LIN {X 0,Y 474.618,Z 134.358,A -85,B 0,C 180,E1 -7419.646,E2 -7419.646} C_VEL
LIN {X 0,Y 474.617,Z 134.363,A -85,B 0,C 180,E1 -7422.934,E2 -7422.934} C_VEL
LIN {X 0,Y 474.606,Z 134.364,A -85,B 0,C 180,E1 -7425.894,E2 -7425.894} C_VEL
LIN {X 0,Y 474.625,Z 134.361,A -85,B 0,C 180,E1 -7429.042,E2 -7429.042} C_VEL
LIN {X 0,Y 474.614,Z 134.364,A -85,B 0,C 180,E1 -7431.704,E2 -7431.704} C_VEL
LIN {X 0,Y 474.628,Z 134.361,A -85,B 0,C 180,E1 -7434.726,E2 -7434.726} C_VEL
LIN {X 0,Y 474.64,Z 134.365,A -85,B 0,C 180,E1 -7437.788,E2 -7437.788} C_VEL
LIN {X 0,Y 474.627,Z 134.362,A -85,B 0,C 180,E1 -7440.885,E2 -7440.885} C_VEL
LIN {X 0,Y 474.666,Z 134.362,A -85,B 0,C 180,E1 -7443.628,E2 -7443.628} C_VEL
LIN {X 0,Y 474.697,Z 134.422,A -85,B 0,C 180,E1 -7444.926,E2 -7444.926} C_VEL
LIN {X 0,Y 475.746,Z 140.895,A -85,B 0,C 180,E1 -7446.335,E2 -7446.335} C_VEL
LIN {X 0,Y 475.555,Z 150.09,A -85,B 0,C 180,E1 -7448.214,E2 -7448.214} C_VEL
LIN {X 0,Y 478.426,Z 164.474,A -85,B 0,C 180,E1 -7448.557,E2 -7448.557} C_VEL
LIN {X 0,Y 478.376,Z 175.483,A -85,B 0,C 180,E1 -7448.726,E2 -7448.726} C_VEL
LIN {X 0,Y 477.685,Z 181.33,A -85,B 0,C 180,E1 -7448.79,E2 -7448.79} C_VEL
LIN {X 0,Y 472.03,Z 200.344,A -85,B 0,C 180,E1 -7448.866,E2 -7448.866} C_VEL
LIN {X 0,Y 471.362,Z 206.19,A -85,B 0,C 180,E1 -7448.932,E2 -7448.932} C_VEL
LIN {X 0,Y 470.901,Z 258.071,A -85,B 0,C 180,E1 -7449.753,E2 -7449.753} C_VEL
LIN {X 0,Y 470.549,Z 271.601,A -85,B 0,C 180,E1 -7450.149,E2 -7450.149} C_VEL
LIN {X 0,Y 470.242,Z 283.825,A -85,B 0,C 180,E1 -7450.685,E2 -7450.685} C_VEL
LIN {X 0,Y 469.795,Z 295.138,A -85,B 0,C 180,E1 -7451.351,E2 -7451.351} C_VEL
LIN {X 0,Y 469.182,Z 306.762,A -85,B 0,C 180,E1 -7452.229,E2 -7452.229} C_VEL
LIN {X 0,Y 468.729,Z 317.2,A -85,B 0,C 180,E1 -7453.224,E2 -7453.224} C_VEL
LIN {X 0,Y 468.335,Z 326.528,A -85,B 0,C 180,E1 -7454.328,E2 -7454.328} C_VEL
LIN {X 0,Y 467.799,Z 335.532,A -85,B 0,C 180,E1 -7455.647,E2 -7455.647} C_VEL
LIN {X 0,Y 467.428,Z 342.757,A -85,B 0,C 180,E1 -7456.965,E2 -7456.965} C_VEL
LIN {X 0,Y 467.168,Z 348.535,A -85,B 0,C 180,E1 -7458.293,E2 -7458.293} C_VEL
LIN {X 0,Y 466.955,Z 352.989,A -85,B 0,C 180,E1 -7459.594,E2 -7459.594} C_VEL
LIN {X 0,Y 466.832,Z 355.353,A -85,B 0,C 180,E1 -7460.467,E2 -7460.467} C_VEL
LIN {X 0,Y 466.795,Z 357.283,A -85,B 0,C 180,E1 -7461.34,E2 -7461.34} C_VEL
LIN {X 0,Y 466.753,Z 358.793,A -85,B 0,C 180,E1 -7462.211,E2 -7462.211} C_VEL
LIN {X 0,Y 466.786,Z 360.292,A -85,B 0,C 180,E1 -7463.571,E2 -7463.571} C_VEL
LIN {X 0,Y 466.71,Z 360.795,A -85,B 0,C 180,E1 -7464.815,E2 -7464.815} C_VEL
LIN {X 0,Y 466.671,Z 360.695,A -85,B 0,C 180,E1 -7465.681,E2 -7465.681} C_VEL
LIN {X 0,Y 466.773,Z 360.159,A -85,B 0,C 180,E1 -7466.546,E2 -7466.546} C_VEL
LIN {X 0,Y 466.71,Z 357.94,A -85,B 0,C 180,E1 -7468.273,E2 -7468.273} C_VEL
LIN {X 0,Y 466.756,Z 355.182,A -85,B 0,C 180,E1 -7469.568,E2 -7469.568} C_VEL
LIN {X 0,Y 466.822,Z 351.423,A -85,B 0,C 180,E1 -7470.862,E2 -7470.862} C_VEL
LIN {X 0,Y 467.123,Z 346.544,A -85,B 0,C 180,E1 -7472.155,E2 -7472.155} C_VEL
LIN {X 0,Y 467.282,Z 340.432,A -85,B 0,C 180,E1 -7473.448,E2 -7473.448} C_VEL
LIN {X 0,Y 467.539,Z 335.515,A -85,B 0,C 180,E1 -7474.31,E2 -7474.31} C_VEL
LIN {X 0,Y 468.082,Z 326.668,A -85,B 0,C 180,E1 -7475.6,E2 -7475.6} C_VEL
LIN {X 0,Y 468.554,Z 317.59,A -85,B 0,C 180,E1 -7476.675,E2 -7476.675} C_VEL
LIN {X 0,Y 469.073,Z 307.492,A -85,B 0,C 180,E1 -7477.64,E2 -7477.64} C_VEL
LIN {X 0,Y 469.554,Z 296.307,A -85,B 0,C 180,E1 -7478.499,E2 -7478.499} C_VEL
LIN {X 0,Y 469.933,Z 284.157,A -85,B 0,C 180,E1 -7479.228,E2 -7479.228} C_VEL
LIN {X 0,Y 470.209,Z 271.377,A -85,B 0,C 180,E1 -7479.788,E2 -7479.788} C_VEL
LIN {X 0,Y 470.485,Z 258.684,A -85,B 0,C 180,E1 -7480.162,E2 -7480.162} C_VEL
LIN {X 0,Y 470.775,Z 232.471,A -85,B 0,C 180,E1 -7480.591,E2 -7480.591} C_VEL
LIN {X 0,Y 471.136,Z 164.035,A -85,B 0,C 180,E1 -7481.638,E2 -7481.638} C_VEL
LIN {X 0,Y 468.426,Z 150.239,A -85,B 0,C 180,E1 -7481.96,E2 -7481.96} C_VEL
LIN {X 0,Y 468.453,Z 139.769,A -85,B 0,C 180,E1 -7484.109,E2 -7484.109} C_VEL
LIN {X 0,Y 467.712,Z 135.226,A -85,B 0,C 180,E1 -7485.133,E2 -7485.133} C_VEL
LIN {X 0,Y 467.614,Z 135.236,A -85,B 0,C 180,E1 -7488.762,E2 -7488.762} C_VEL
LIN {X 0,Y 467.581,Z 135.237,A -85,B 0,C 180,E1 -7491.267,E2 -7491.267} C_VEL
LIN {X 0,Y 467.563,Z 135.244,A -85,B 0,C 180,E1 -7493.943,E2 -7493.943} C_VEL
LIN {X 0,Y 467.612,Z 135.235,A -85,B 0,C 180,E1 -7496.799,E2 -7496.799} C_VEL
LIN {X 0,Y 467.551,Z 135.245,A -85,B 0,C 180,E1 -7499.737,E2 -7499.737} C_VEL
LIN {X 0,Y 467.581,Z 135.238,A -85,B 0,C 180,E1 -7502.757,E2 -7502.757} C_VEL
LIN {X 0,Y 467.55,Z 135.249,A -85,B 0,C 180,E1 -7505.888,E2 -7505.888} C_VEL
LIN {X 0,Y 467.578,Z 135.24,A -85,B 0,C 180,E1 -7509.143,E2 -7509.143} C_VEL
LIN {X 0,Y 467.581,Z 135.239,A -85,B 0,C 180,E1 -7512.566,E2 -7512.566} C_VEL
LIN {X 0,Y 467.56,Z 135.243,A -85,B 0,C 180,E1 -7515.051,E2 -7515.051} C_VEL
LIN {X 0,Y 467.582,Z 135.243,A -85,B 0,C 180,E1 -7517.439,E2 -7517.439} C_VEL
LIN {X 0,Y 467.552,Z 135.244,A -85,B 0,C 180,E1 -7520.852,E2 -7520.852} C_VEL
LIN {X 0,Y 467.55,Z 135.243,A -85,B 0,C 180,E1 -7524.26,E2 -7524.26} C_VEL
LIN {X 0,Y 467.57,Z 135.245,A -85,B 0,C 180,E1 -7527.32,E2 -7527.32} C_VEL
LIN {X 0,Y 467.558,Z 135.244,A -85,B 0,C 180,E1 -7530.667,E2 -7530.667} C_VEL
LIN {X 0,Y 467.576,Z 135.244,A -85,B 0,C 180,E1 -7533.197,E2 -7533.197} C_VEL
LIN {X 0,Y 467.578,Z 135.241,A -85,B 0,C 180,E1 -7536.469,E2 -7536.469} C_VEL
LIN {X 0,Y 467.609,Z 135.237,A -85,B 0,C 180,E1 -7539.776,E2 -7539.776} C_VEL
LIN {X 0,Y 467.575,Z 135.242,A -85,B 0,C 180,E1 -7542.505,E2 -7542.505} C_VEL
LIN {X 0,Y 467.584,Z 135.24,A -85,B 0,C 180,E1 -7545.196,E2 -7545.196} C_VEL
LIN {X 0,Y 467.644,Z 135.234,A -85,B 0,C 180,E1 -7547.854,E2 -7547.854} C_VEL
LIN {X 0,Y 467.653,Z 135.231,A -85,B 0,C 180,E1 -7551.357,E2 -7551.357} C_VEL
LIN {X 0,Y 467.69,Z 135.228,A -85,B 0,C 180,E1 -7553.962,E2 -7553.962} C_VEL
LIN {X 0,Y 467.799,Z 135.214,A -85,B 0,C 180,E1 -7557.417,E2 -7557.417} C_VEL
LIN {X 0,Y 467.836,Z 135.21,A -85,B 0,C 180,E1 -7560,E2 -7560} C_VEL
LIN {X 0,Y 467.8,Z 135.214,A -85,B 0,C 180,E1 -7562.583,E2 -7562.583} C_VEL
LIN {X 0,Y 467.695,Z 135.227,A -85,B 0,C 180,E1 -7566.038,E2 -7566.038} C_VEL
LIN {X 0,Y 467.653,Z 135.231,A -85,B 0,C 180,E1 -7568.643,E2 -7568.643} C_VEL
LIN {X 0,Y 467.644,Z 135.234,A -85,B 0,C 180,E1 -7572.146,E2 -7572.146} C_VEL
LIN {X 0,Y 467.636,Z 135.234,A -85,B 0,C 180,E1 -7575.885,E2 -7575.885} C_VEL
LIN {X 0,Y 467.609,Z 135.238,A -85,B 0,C 180,E1 -7579.308,E2 -7579.308} C_VEL
LIN {X 0,Y 467.519,Z 135.248,A -85,B 0,C 180,E1 -7582.075,E2 -7582.075} C_VEL
LIN {X 0,Y 467.557,Z 135.247,A -85,B 0,C 180,E1 -7584.89,E2 -7584.89} C_VEL
LIN {X 0,Y 467.605,Z 135.237,A -85,B 0,C 180,E1 -7587.77,E2 -7587.77} C_VEL
LIN {X 0,Y 467.557,Z 135.245,A -85,B 0,C 180,E1 -7591.045,E2 -7591.045} C_VEL
LIN {X 0,Y 467.567,Z 135.242,A -85,B 0,C 180,E1 -7594.241,E2 -7594.241} C_VEL
LIN {X 0,Y 467.538,Z 135.245,A -85,B 0,C 180,E1 -7597.187,E2 -7597.187} C_VEL
LIN {X 0,Y 467.566,Z 135.244,A -85,B 0,C 180,E1 -7600.266,E2 -7600.266} C_VEL
LIN {X 0,Y 467.579,Z 135.243,A -85,B 0,C 180,E1 -7602.568,E2 -7602.568} C_VEL
LIN {X 0,Y 467.559,Z 135.242,A -85,B 0,C 180,E1 -7605.054,E2 -7605.054} C_VEL
LIN {X 0,Y 467.583,Z 135.238,A -85,B 0,C 180,E1 -7607.441,E2 -7607.441} C_VEL
LIN {X 0,Y 467.577,Z 135.239,A -85,B 0,C 180,E1 -7610.856,E2 -7610.856} C_VEL
LIN {X 0,Y 467.555,Z 135.246,A -85,B 0,C 180,E1 -7614.262,E2 -7614.262} C_VEL
LIN {X 0,Y 467.578,Z 135.238,A -85,B 0,C 180,E1 -7617.322,E2 -7617.322} C_VEL
LIN {X 0,Y 467.567,Z 135.243,A -85,B 0,C 180,E1 -7620.669,E2 -7620.669} C_VEL
LIN {X 0,Y 467.651,Z 135.252,A -85,B 0,C 180,E1 -7623.714,E2 -7623.714} C_VEL
LIN {X 0,Y 469.785,Z 147.105,A -85,B 0,C 180,E1 -7625.862,E2 -7625.862} C_VEL
LIN {X 0,Y 469.132,Z 164.184,A -85,B 0,C 180,E1 -7628.742,E2 -7628.742} C_VEL
LIN {X 0,Y 468.427,Z 182.92,A -85,B 0,C 180,E1 -7631.862,E2 -7631.862} C_VEL
LIN {X 0,Y 468.193,Z 190.165,A -85,B 0,C 180,E1 -7633.061,E2 -7633.061} C_VEL
LIN {X 0,Y 471.01,Z 210.369,A -85,B 0,C 180,E1 -7633.47,E2 -7633.47} C_VEL
LIN {X 0,Y 470.392,Z 299.136,A -85,B 0,C 180,E1 -7634.844,E2 -7634.844} C_VEL
LIN {X 0,Y 469.994,Z 311.574,A -85,B 0,C 180,E1 -7635.191,E2 -7635.191} C_VEL
LIN {X 0,Y 469.516,Z 325.058,A -85,B 0,C 180,E1 -7635.757,E2 -7635.757} C_VEL
LIN {X 0,Y 469.017,Z 337.151,A -85,B 0,C 180,E1 -7636.46,E2 -7636.46} C_VEL
LIN {X 0,Y 468.525,Z 348.652,A -85,B 0,C 180,E1 -7637.324,E2 -7637.324} C_VEL
LIN {X 0,Y 468.07,Z 359.11,A -85,B 0,C 180,E1 -7638.306,E2 -7638.306} C_VEL
LIN {X 0,Y 467.602,Z 368.448,A -85,B 0,C 180,E1 -7639.391,E2 -7639.391} C_VEL
LIN {X 0,Y 467.207,Z 377.51,A -85,B 0,C 180,E1 -7640.695,E2 -7640.695} C_VEL
LIN {X 0,Y 466.979,Z 384.813,A -85,B 0,C 180,E1 -7641.999,E2 -7641.999} C_VEL
LIN {X 0,Y 466.827,Z 389.743,A -85,B 0,C 180,E1 -7643.083,E2 -7643.083} C_VEL
LIN {X 0,Y 466.749,Z 394.534,A -85,B 0,C 180,E1 -7644.384,E2 -7644.384} C_VEL
LIN {X 0,Y 466.647,Z 398.195,A -85,B 0,C 180,E1 -7645.682,E2 -7645.682} C_VEL
LIN {X 0,Y 466.73,Z 400.093,A -85,B 0,C 180,E1 -7646.548,E2 -7646.548} C_VEL
LIN {X 0,Y 466.685,Z 401.519,A -85,B 0,C 180,E1 -7647.411,E2 -7647.411} C_VEL
LIN {X 0,Y 466.662,Z 402.532,A -85,B 0,C 180,E1 -7648.275,E2 -7648.275} C_VEL
LIN {X 0,Y 466.611,Z 403.387,A -85,B 0,C 180,E1 -7650.001,E2 -7650.001} C_VEL
LIN {X 0,Y 466.627,Z 403.192,A -85,B 0,C 180,E1 -7650.864,E2 -7650.864} C_VEL
LIN {X 0,Y 466.662,Z 402.596,A -85,B 0,C 180,E1 -7651.727,E2 -7651.727} C_VEL
LIN {X 0,Y 466.685,Z 401.61,A -85,B 0,C 180,E1 -7652.59,E2 -7652.59} C_VEL
LIN {X 0,Y 466.7,Z 400.226,A -85,B 0,C 180,E1 -7653.454,E2 -7653.454} C_VEL
LIN {X 0,Y 466.687,Z 397.304,A -85,B 0,C 180,E1 -7654.752,E2 -7654.752} C_VEL
LIN {X 0,Y 466.719,Z 393.351,A -85,B 0,C 180,E1 -7656.051,E2 -7656.051} C_VEL
LIN {X 0,Y 466.883,Z 388.271,A -85,B 0,C 180,E1 -7657.352,E2 -7657.352} C_VEL
LIN {X 0,Y 467.112,Z 381.892,A -85,B 0,C 180,E1 -7658.654,E2 -7658.654} C_VEL
LIN {X 0,Y 467.425,Z 373.921,A -85,B 0,C 180,E1 -7659.958,E2 -7659.958} C_VEL
LIN {X 0,Y 467.878,Z 365.819,A -85,B 0,C 180,E1 -7661.042,E2 -7661.042} C_VEL
LIN {X 0,Y 468.324,Z 355.951,A -85,B 0,C 180,E1 -7662.128,E2 -7662.128} C_VEL
LIN {X 0,Y 468.809,Z 344.917,A -85,B 0,C 180,E1 -7663.106,E2 -7663.106} C_VEL
LIN {X 0,Y 469.352,Z 334.121,A -85,B 0,C 180,E1 -7663.862,E2 -7663.862} C_VEL
LIN {X 0,Y 469.895,Z 321.117,A -85,B 0,C 180,E1 -7664.564,E2 -7664.564} C_VEL
LIN {X 0,Y 470.368,Z 308.577,A -85,B 0,C 180,E1 -7665.047,E2 -7665.047} C_VEL
LIN {X 0,Y 470.732,Z 295.474,A -85,B 0,C 180,E1 -7665.368,E2 -7665.368} C_VEL
LIN {X 0,Y 471.218,Z 209.135,A -85,B 0,C 180,E1 -7666.708,E2 -7666.708} C_VEL
LIN {X 0,Y 468.32,Z 189.921,A -85,B 0,C 180,E1 -7667.145,E2 -7667.145} C_VEL
LIN {X 0,Y 468.918,Z 173.306,A -85,B 0,C 180,E1 -7669.937,E2 -7669.937} C_VEL
LIN {X 0,Y 469.766,Z 155.911,A -85,B 0,C 180,E1 -7672.891,E2 -7672.891} C_VEL
LIN {X 0,Y 469.986,Z 147.08,A -85,B 0,C 180,E1 -7674.421,E2 -7674.421} C_VEL
LIN {X 0,Y 467.614,Z 135.239,A -85,B 0,C 180,E1 -7676.68,E2 -7676.68} C_VEL
LIN {X 0,Y 467.55,Z 135.251,A -85,B 0,C 180,E1 -7679.739,E2 -7679.739} C_VEL
LIN {X 0,Y 467.586,Z 135.24,A -85,B 0,C 180,E1 -7682.759,E2 -7682.759} C_VEL
LIN {X 0,Y 467.553,Z 135.246,A -85,B 0,C 180,E1 -7685.89,E2 -7685.89} C_VEL
LIN {X 0,Y 467.557,Z 135.242,A -85,B 0,C 180,E1 -7689.148,E2 -7689.148} C_VEL
LIN {X 0,Y 467.575,Z 135.243,A -85,B 0,C 180,E1 -7691.403,E2 -7691.403} C_VEL
LIN {X 0,Y 467.567,Z 135.242,A -85,B 0,C 180,E1 -7695.052,E2 -7695.052} C_VEL
LIN {X 0,Y 467.568,Z 135.24,A -85,B 0,C 180,E1 -7698.596,E2 -7698.596} C_VEL
LIN {X 0,Y 467.564,Z 135.241,A -85,B 0,C 180,E1 -7701.955,E2 -7701.955} C_VEL
LIN {X 0,Y 467.559,Z 135.247,A -85,B 0,C 180,E1 -7705.167,E2 -7705.167} C_VEL
LIN {X 0,Y 467.58,Z 135.239,A -85,B 0,C 180,E1 -7708.26,E2 -7708.26} C_VEL
LIN {X 0,Y 467.544,Z 135.245,A -85,B 0,C 180,E1 -7711.248,E2 -7711.248} C_VEL
LIN {X 0,Y 467.578,Z 135.24,A -85,B 0,C 180,E1 -7714.401,E2 -7714.401} C_VEL
LIN {X 0,Y 467.568,Z 135.243,A -85,B 0,C 180,E1 -7716.995,E2 -7716.995} C_VEL
LIN {X 0,Y 467.61,Z 135.231,A -85,B 0,C 180,E1 -7719.777,E2 -7719.777} C_VEL
LIN {X 0,Y 467.564,Z 135.245,A -85,B 0,C 180,E1 -7722.505,E2 -7722.505} C_VEL
LIN {X 0,Y 467.586,Z 135.232,A -85,B 0,C 180,E1 -7725.196,E2 -7725.196} C_VEL
LIN {X 0,Y 467.64,Z 135.231,A -85,B 0,C 180,E1 -7727.854,E2 -7727.854} C_VEL
LIN {X 0,Y 467.628,Z 135.226,A -85,B 0,C 180,E1 -7731.356,E2 -7731.356} C_VEL
LIN {X 0,Y 467.698,Z 135.228,A -85,B 0,C 180,E1 -7733.962,E2 -7733.962} C_VEL
LIN {X 0,Y 467.808,Z 135.205,A -85,B 0,C 180,E1 -7737.417,E2 -7737.417} C_VEL
LIN {X 0,Y 467.848,Z 135.21,A -85,B 0,C 180,E1 -7740,E2 -7740} C_VEL
LIN {X 0,Y 467.811,Z 135.203,A -85,B 0,C 180,E1 -7742.583,E2 -7742.583} C_VEL
LIN {X 0,Y 467.7,Z 135.226,A -85,B 0,C 180,E1 -7746.038,E2 -7746.038} C_VEL
LIN {X 0,Y 467.663,Z 135.221,A -85,B 0,C 180,E1 -7748.643,E2 -7748.643} C_VEL
LIN {X 0,Y 467.656,Z 135.228,A -85,B 0,C 180,E1 -7752.146,E2 -7752.146} C_VEL
LIN {X 0,Y 467.649,Z 135.23,A -85,B 0,C 180,E1 -7755.885,E2 -7755.885} C_VEL
LIN {X 0,Y 467.621,Z 135.234,A -85,B 0,C 180,E1 -7759.308,E2 -7759.308} C_VEL
LIN {X 0,Y 467.531,Z 135.244,A -85,B 0,C 180,E1 -7762.074,E2 -7762.074} C_VEL
LIN {X 0,Y 467.569,Z 135.24,A -85,B 0,C 180,E1 -7764.89,E2 -7764.89} C_VEL
LIN {X 0,Y 467.581,Z 135.236,A -85,B 0,C 180,E1 -7767.772,E2 -7767.772} C_VEL
LIN {X 0,Y 467.568,Z 135.243,A -85,B 0,C 180,E1 -7771.045,E2 -7771.045} C_VEL
LIN {X 0,Y 467.579,Z 135.239,A -85,B 0,C 180,E1 -7774.24,E2 -7774.24} C_VEL
LIN {X 0,Y 467.549,Z 135.243,A -85,B 0,C 180,E1 -7777.186,E2 -7777.186} C_VEL
LIN {X 0,Y 467.577,Z 135.238,A -85,B 0,C 180,E1 -7780.265,E2 -7780.265} C_VEL
LIN {X 0,Y 467.59,Z 135.239,A -85,B 0,C 180,E1 -7782.567,E2 -7782.567} C_VEL
LIN {X 0,Y 467.568,Z 135.239,A -85,B 0,C 180,E1 -7785.053,E2 -7785.053} C_VEL
LIN {X 0,Y 467.576,Z 135.242,A -85,B 0,C 180,E1 -7788.597,E2 -7788.597} C_VEL
LIN {X 0,Y 467.564,Z 135.24,A -85,B 0,C 180,E1 -7791.409,E2 -7791.409} C_VEL
LIN {X 0,Y 467.564,Z 135.245,A -85,B 0,C 180,E1 -7794.261,E2 -7794.261} C_VEL
LIN {X 0,Y 467.586,Z 135.239,A -85,B 0,C 180,E1 -7797.321,E2 -7797.321} C_VEL
LIN {X 0,Y 467.573,Z 135.241,A -85,B 0,C 180,E1 -7800.668,E2 -7800.668} C_VEL
LIN {X 0,Y 467.621,Z 135.238,A -85,B 0,C 180,E1 -7803.2,E2 -7803.2} C_VEL
LIN {X 0,Y 467.657,Z 135.37,A -85,B 0,C 180,E1 -7804.742,E2 -7804.742} C_VEL
LIN {X 0,Y 468.808,Z 142.348,A -85,B 0,C 180,E1 -7806.277,E2 -7806.277} C_VEL
LIN {X 0,Y 468.64,Z 150.392,A -85,B 0,C 180,E1 -7807.937,E2 -7807.937} C_VEL
LIN {X 0,Y 471.683,Z 165.079,A -85,B 0,C 180,E1 -7808.299,E2 -7808.299} C_VEL
LIN {X 0,Y 471.362,Z 206.19,A -85,B 0,C 180,E1 -7808.932,E2 -7808.932} C_VEL
LIN {X 0,Y 470.683,Z 212.035,A -85,B 0,C 180,E1 -7808.997,E2 -7808.997} C_VEL
LIN {X 0,Y 464.988,Z 231.034,A -85,B 0,C 180,E1 -7809.074,E2 -7809.074} C_VEL
LIN {X 0,Y 464.348,Z 236.877,A -85,B 0,C 180,E1 -7809.142,E2 -7809.142} C_VEL
LIN {X 0,Y 464.074,Z 259.518,A -85,B 0,C 180,E1 -7809.528,E2 -7809.528} C_VEL
LIN {X 0,Y 463.761,Z 272.58,A -85,B 0,C 180,E1 -7809.929,E2 -7809.929} C_VEL
LIN {X 0,Y 463.436,Z 283.39,A -85,B 0,C 180,E1 -7810.41,E2 -7810.41} C_VEL
LIN {X 0,Y 462.994,Z 294.64,A -85,B 0,C 180,E1 -7811.067,E2 -7811.067} C_VEL
LIN {X 0,Y 462.342,Z 306.423,A -85,B 0,C 180,E1 -7811.957,E2 -7811.957} C_VEL
LIN {X 0,Y 461.893,Z 316.974,A -85,B 0,C 180,E1 -7812.968,E2 -7812.968} C_VEL
LIN {X 0,Y 461.402,Z 326.432,A -85,B 0,C 180,E1 -7814.087,E2 -7814.087} C_VEL
LIN {X 0,Y 460.835,Z 335.506,A -85,B 0,C 180,E1 -7815.425,E2 -7815.425} C_VEL
LIN {X 0,Y 460.428,Z 342.792,A -85,B 0,C 180,E1 -7816.763,E2 -7816.763} C_VEL
LIN {X 0,Y 460.136,Z 348.828,A -85,B 0,C 180,E1 -7818.161,E2 -7818.161} C_VEL
LIN {X 0,Y 459.924,Z 353.147,A -85,B 0,C 180,E1 -7819.433,E2 -7819.433} C_VEL
LIN {X 0,Y 459.764,Z 355.539,A -85,B 0,C 180,E1 -7820.319,E2 -7820.319} C_VEL
LIN {X 0,Y 459.732,Z 357.49,A -85,B 0,C 180,E1 -7821.206,E2 -7821.206} C_VEL
LIN {X 0,Y 459.669,Z 359.028,A -85,B 0,C 180,E1 -7822.09,E2 -7822.09} C_VEL
LIN {X 0,Y 459.715,Z 360.645,A -85,B 0,C 180,E1 -7823.569,E2 -7823.569} C_VEL
LIN {X 0,Y 459.643,Z 361.108,A -85,B 0,C 180,E1 -7824.736,E2 -7824.736} C_VEL
LIN {X 0,Y 459.582,Z 361.034,A -85,B 0,C 180,E1 -7825.614,E2 -7825.614} C_VEL
LIN {X 0,Y 459.699,Z 360.535,A -85,B 0,C 180,E1 -7826.493,E2 -7826.493} C_VEL
LIN {X 0,Y 459.647,Z 358.356,A -85,B 0,C 180,E1 -7828.247,E2 -7828.247} C_VEL
LIN {X 0,Y 459.669,Z 355.644,A -85,B 0,C 180,E1 -7829.561,E2 -7829.561} C_VEL
LIN {X 0,Y 459.745,Z 351.931,A -85,B 0,C 180,E1 -7830.875,E2 -7830.875} C_VEL
LIN {X 0,Y 460.067,Z 347.1,A -85,B 0,C 180,E1 -7832.188,E2 -7832.188} C_VEL
LIN {X 0,Y 460.234,Z 341.041,A -85,B 0,C 180,E1 -7833.501,E2 -7833.501} C_VEL
LIN {X 0,Y 460.707,Z 333.493,A -85,B 0,C 180,E1 -7834.812,E2 -7834.812} C_VEL
LIN {X 0,Y 461.228,Z 324.015,A -85,B 0,C 180,E1 -7836.122,E2 -7836.122} C_VEL
LIN {X 0,Y 461.803,Z 314.239,A -85,B 0,C 180,E1 -7837.212,E2 -7837.212} C_VEL
LIN {X 0,Y 462.333,Z 303.269,A -85,B 0,C 180,E1 -7838.192,E2 -7838.192} C_VEL
LIN {X 0,Y 462.81,Z 291.752,A -85,B 0,C 180,E1 -7839.003,E2 -7839.003} C_VEL
LIN {X 0,Y 463.181,Z 279.605,A -85,B 0,C 180,E1 -7839.662,E2 -7839.662} C_VEL
LIN {X 0,Y 463.481,Z 266.996,A -85,B 0,C 180,E1 -7840.152,E2 -7840.152} C_VEL
LIN {X 0,Y 463.673,Z 253.728,A -85,B 0,C 180,E1 -7840.479,E2 -7840.479} C_VEL
LIN {X 0,Y 464.349,Z 165.216,A -85,B 0,C 180,E1 -7841.853,E2 -7841.853} C_VEL
LIN {X 0,Y 461.447,Z 150.541,A -85,B 0,C 180,E1 -7842.199,E2 -7842.199} C_VEL
LIN {X 0,Y 461.511,Z 141.339,A -85,B 0,C 180,E1 -7844.101,E2 -7844.101} C_VEL
LIN {X 0,Y 460.668,Z 136.104,A -85,B 0,C 180,E1 -7845.257,E2 -7845.257} C_VEL
LIN {X 0,Y 460.568,Z 136.112,A -85,B 0,C 180,E1 -7848.899,E2 -7848.899} C_VEL
LIN {X 0,Y 460.516,Z 136.118,A -85,B 0,C 180,E1 -7851.484,E2 -7851.484} C_VEL
LIN {X 0,Y 460.531,Z 136.121,A -85,B 0,C 180,E1 -7854.332,E2 -7854.332} C_VEL
LIN {X 0,Y 460.57,Z 136.112,A -85,B 0,C 180,E1 -7857.243,E2 -7857.243} C_VEL
LIN {X 0,Y 460.508,Z 136.123,A -85,B 0,C 180,E1 -7860.239,E2 -7860.239} C_VEL
LIN {X 0,Y 460.526,Z 136.118,A -85,B 0,C 180,E1 -7863.324,E2 -7863.324} C_VEL
LIN {X 0,Y 460.472,Z 136.125,A -85,B 0,C 180,E1 -7866.528,E2 -7866.528} C_VEL
LIN {X 0,Y 460.553,Z 136.119,A -85,B 0,C 180,E1 -7869.858,E2 -7869.858} C_VEL
LIN {X 0,Y 460.507,Z 136.121,A -85,B 0,C 180,E1 -7872.899,E2 -7872.899} C_VEL
LIN {X 0,Y 460.501,Z 136.124,A -85,B 0,C 180,E1 -7875.83,E2 -7875.83} C_VEL
LIN {X 0,Y 460.523,Z 136.119,A -85,B 0,C 180,E1 -7878.988,E2 -7878.988} C_VEL
LIN {X 0,Y 460.511,Z 136.123,A -85,B 0,C 180,E1 -7881.265,E2 -7881.265} C_VEL
LIN {X 0,Y 460.5,Z 136.123,A -85,B 0,C 180,E1 -7884.553,E2 -7884.553} C_VEL
LIN {X 0,Y 460.52,Z 136.12,A -85,B 0,C 180,E1 -7887.714,E2 -7887.714} C_VEL
LIN {X 0,Y 460.528,Z 136.119,A -85,B 0,C 180,E1 -7890.768,E2 -7890.768} C_VEL
LIN {X 0,Y 460.531,Z 136.118,A -85,B 0,C 180,E1 -7893.733,E2 -7893.733} C_VEL
LIN {X 0,Y 460.531,Z 136.119,A -85,B 0,C 180,E1 -7896.623,E2 -7896.623} C_VEL
LIN {X 0,Y 460.538,Z 136.118,A -85,B 0,C 180,E1 -7899.452,E2 -7899.452} C_VEL
LIN {X 0,Y 460.528,Z 136.12,A -85,B 0,C 180,E1 -7902.229,E2 -7902.229} C_VEL
LIN {X 0,Y 460.545,Z 136.119,A -85,B 0,C 180,E1 -7904.964,E2 -7904.964} C_VEL
LIN {X 0,Y 460.596,Z 136.112,A -85,B 0,C 180,E1 -7908.559,E2 -7908.559} C_VEL
LIN {X 0,Y 460.604,Z 136.11,A -85,B 0,C 180,E1 -7911.223,E2 -7911.223} C_VEL
LIN {X 0,Y 460.656,Z 136.104,A -85,B 0,C 180,E1 -7913.869,E2 -7913.869} C_VEL
LIN {X 0,Y 460.743,Z 136.093,A -85,B 0,C 180,E1 -7917.377,E2 -7917.377} C_VEL
LIN {X 0,Y 460.805,Z 136.085,A -85,B 0,C 180,E1 -7920,E2 -7920} C_VEL
LIN {X 0,Y 460.744,Z 136.093,A -85,B 0,C 180,E1 -7922.623,E2 -7922.623} C_VEL
LIN {X 0,Y 460.661,Z 136.103,A -85,B 0,C 180,E1 -7926.13,E2 -7926.13} C_VEL
LIN {X 0,Y 460.604,Z 136.109,A -85,B 0,C 180,E1 -7928.777,E2 -7928.777} C_VEL
LIN {X 0,Y 460.584,Z 136.112,A -85,B 0,C 180,E1 -7932.435,E2 -7932.435} C_VEL
LIN {X 0,Y 460.589,Z 136.112,A -85,B 0,C 180,E1 -7935.998,E2 -7935.998} C_VEL
LIN {X 0,Y 460.555,Z 136.116,A -85,B 0,C 180,E1 -7939.616,E2 -7939.616} C_VEL
LIN {X 0,Y 460.495,Z 136.123,A -85,B 0,C 180,E1 -7942.429,E2 -7942.429} C_VEL
LIN {X 0,Y 460.535,Z 136.118,A -85,B 0,C 180,E1 -7945.797,E2 -7945.797} C_VEL
LIN {X 0,Y 460.539,Z 136.117,A -85,B 0,C 180,E1 -7948.234,E2 -7948.234} C_VEL
LIN {X 0,Y 460.51,Z 136.121,A -85,B 0,C 180,E1 -7951.283,E2 -7951.283} C_VEL
LIN {X 0,Y 460.513,Z 136.123,A -85,B 0,C 180,E1 -7954.505,E2 -7954.505} C_VEL
LIN {X 0,Y 460.492,Z 136.122,A -85,B 0,C 180,E1 -7957.624,E2 -7957.624} C_VEL
LIN {X 0,Y 460.531,Z 136.12,A -85,B 0,C 180,E1 -7960.27,E2 -7960.27} C_VEL
LIN {X 0,Y 460.489,Z 136.122,A -85,B 0,C 180,E1 -7963.377,E2 -7963.377} C_VEL
LIN {X 0,Y 460.492,Z 136.124,A -85,B 0,C 180,E1 -7966.626,E2 -7966.626} C_VEL
LIN {X 0,Y 460.536,Z 136.117,A -85,B 0,C 180,E1 -7969.732,E2 -7969.732} C_VEL
LIN {X 0,Y 460.494,Z 136.123,A -85,B 0,C 180,E1 -7972.525,E2 -7972.525} C_VEL
LIN {X 0,Y 460.542,Z 136.116,A -85,B 0,C 180,E1 -7975.625,E2 -7975.625} C_VEL
LIN {X 0,Y 460.534,Z 136.118,A -85,B 0,C 180,E1 -7978.746,E2 -7978.746} C_VEL
LIN {X 0,Y 460.579,Z 136.115,A -85,B 0,C 180,E1 -7982.255,E2 -7982.255} C_VEL
LIN {X 0,Y 460.618,Z 136.308,A -85,B 0,C 180,E1 -7983.556,E2 -7983.556} C_VEL
LIN {X 0,Y 462.777,Z 147.763,A -85,B 0,C 180,E1 -7985.671,E2 -7985.671} C_VEL
LIN {X 0,Y 462.29,Z 161.486,A -85,B 0,C 180,E1 -7988.027,E2 -7988.027} C_VEL
LIN {X 0,Y 461.531,Z 181.108,A -85,B 0,C 180,E1 -7991.352,E2 -7991.352} C_VEL
LIN {X 0,Y 461.196,Z 189.853,A -85,B 0,C 180,E1 -7992.821,E2 -7992.821} C_VEL
LIN {X 0,Y 464.146,Z 211.204,A -85,B 0,C 180,E1 -7993.258,E2 -7993.258} C_VEL
LIN {X 0,Y 463.508,Z 299.121,A -85,B 0,C 180,E1 -7994.642,E2 -7994.642} C_VEL
LIN {X 0,Y 463.061,Z 312.224,A -85,B 0,C 180,E1 -7995.021,E2 -7995.021} C_VEL
LIN {X 0,Y 462.627,Z 324.325,A -85,B 0,C 180,E1 -7995.541,E2 -7995.541} C_VEL
LIN {X 0,Y 462.057,Z 336.54,A -85,B 0,C 180,E1 -7996.253,E2 -7996.253} C_VEL
LIN {X 0,Y 461.533,Z 348.094,A -85,B 0,C 180,E1 -7997.129,E2 -7997.129} C_VEL
LIN {X 0,Y 461.052,Z 358.597,A -85,B 0,C 180,E1 -7998.126,E2 -7998.126} C_VEL
LIN {X 0,Y 460.594,Z 367.984,A -85,B 0,C 180,E1 -7999.228,E2 -7999.228} C_VEL
LIN {X 0,Y 460.163,Z 377.07,A -85,B 0,C 180,E1 -8000.551,E2 -8000.551} C_VEL
LIN {X 0,Y 459.907,Z 384.394,A -85,B 0,C 180,E1 -8001.875,E2 -8001.875} C_VEL
LIN {X 0,Y 459.739,Z 389.343,A -85,B 0,C 180,E1 -8002.976,E2 -8002.976} C_VEL
LIN {X 0,Y 459.645,Z 394.152,A -85,B 0,C 180,E1 -8004.297,E2 -8004.297} C_VEL
LIN {X 0,Y 459.564,Z 397.829,A -85,B 0,C 180,E1 -8005.616,E2 -8005.616} C_VEL
LIN {X 0,Y 459.625,Z 399.735,A -85,B 0,C 180,E1 -8006.494,E2 -8006.494} C_VEL
LIN {X 0,Y 459.607,Z 401.174,A -85,B 0,C 180,E1 -8007.372,E2 -8007.372} C_VEL
LIN {X 0,Y 459.559,Z 402.822,A -85,B 0,C 180,E1 -8009.125,E2 -8009.125} C_VEL
LIN {X 0,Y 459.542,Z 403.062,A -85,B 0,C 180,E1 -8010.001,E2 -8010.001} C_VEL
LIN {X 0,Y 459.56,Z 402.879,A -85,B 0,C 180,E1 -8010.877,E2 -8010.877} C_VEL
LIN {X 0,Y 459.605,Z 401.308,A -85,B 0,C 180,E1 -8012.63,E2 -8012.63} C_VEL
LIN {X 0,Y 459.595,Z 399.93,A -85,B 0,C 180,E1 -8013.508,E2 -8013.508} C_VEL
LIN {X 0,Y 459.614,Z 397.022,A -85,B 0,C 180,E1 -8014.825,E2 -8014.825} C_VEL
LIN {X 0,Y 459.635,Z 392.408,A -85,B 0,C 180,E1 -8016.343,E2 -8016.343} C_VEL
LIN {X 0,Y 459.869,Z 386.034,A -85,B 0,C 180,E1 -8017.906,E2 -8017.906} C_VEL
LIN {X 0,Y 460.15,Z 379.195,A -85,B 0,C 180,E1 -8019.229,E2 -8019.229} C_VEL
LIN {X 0,Y 460.531,Z 370.693,A -85,B 0,C 180,E1 -8020.553,E2 -8020.553} C_VEL
LIN {X 0,Y 461.042,Z 361.963,A -85,B 0,C 180,E1 -8021.653,E2 -8021.653} C_VEL
LIN {X 0,Y 461.532,Z 351.797,A -85,B 0,C 180,E1 -8022.703,E2 -8022.703} C_VEL
LIN {X 0,Y 462.142,Z 340.565,A -85,B 0,C 180,E1 -8023.634,E2 -8023.634} C_VEL
LIN {X 0,Y 462.749,Z 328.631,A -85,B 0,C 180,E1 -8024.401,E2 -8024.401} C_VEL
LIN {X 0,Y 463.292,Z 316.226,A -85,B 0,C 180,E1 -8025.001,E2 -8025.001} C_VEL
LIN {X 0,Y 463.743,Z 303.43,A -85,B 0,C 180,E1 -8025.436,E2 -8025.436} C_VEL
LIN {X 0,Y 463.992,Z 289.871,A -85,B 0,C 180,E1 -8025.709,E2 -8025.709} C_VEL
LIN {X 0,Y 464.516,Z 210.176,A -85,B 0,C 180,E1 -8026.956,E2 -8026.956} C_VEL
LIN {X 0,Y 461.362,Z 189.617,A -85,B 0,C 180,E1 -8027.429,E2 -8027.429} C_VEL
LIN {X 0,Y 462.007,Z 173.117,A -85,B 0,C 180,E1 -8030.248,E2 -8030.248} C_VEL
LIN {X 0,Y 462.859,Z 157.071,A -85,B 0,C 180,E1 -8033.016,E2 -8033.016} C_VEL
LIN {X 0,Y 463.137,Z 149.036,A -85,B 0,C 180,E1 -8034.427,E2 -8034.427} C_VEL
LIN {X 0,Y 460.727,Z 136.92,A -85,B 0,C 180,E1 -8036.744,E2 -8036.744} C_VEL
LIN {X 0,Y 460.584,Z 136.114,A -85,B 0,C 180,E1 -8036.937,E2 -8036.937} C_VEL
LIN {X 0,Y 460.51,Z 136.128,A -85,B 0,C 180,E1 -8040.241,E2 -8040.241} C_VEL
LIN {X 0,Y 460.532,Z 136.12,A -85,B 0,C 180,E1 -8043.325,E2 -8043.325} C_VEL
LIN {X 0,Y 460.475,Z 136.122,A -85,B 0,C 180,E1 -8046.53,E2 -8046.53} C_VEL
LIN {X 0,Y 460.522,Z 136.121,A -85,B 0,C 180,E1 -8049.864,E2 -8049.864} C_VEL
LIN {X 0,Y 460.494,Z 136.12,A -85,B 0,C 180,E1 -8052.898,E2 -8052.898} C_VEL
LIN {X 0,Y 460.506,Z 136.122,A -85,B 0,C 180,E1 -8055.831,E2 -8055.831} C_VEL
LIN {X 0,Y 460.521,Z 136.121,A -85,B 0,C 180,E1 -8058.987,E2 -8058.987} C_VEL
LIN {X 0,Y 460.501,Z 136.12,A -85,B 0,C 180,E1 -8062.377,E2 -8062.377} C_VEL
LIN {X 0,Y 460.537,Z 136.117,A -85,B 0,C 180,E1 -8065.623,E2 -8065.623} C_VEL
LIN {X 0,Y 460.538,Z 136.12,A -85,B 0,C 180,E1 -8068.745,E2 -8068.745} C_VEL
LIN {X 0,Y 460.531,Z 136.116,A -85,B 0,C 180,E1 -8072.266,E2 -8072.266} C_VEL
LIN {X 0,Y 460.522,Z 136.122,A -85,B 0,C 180,E1 -8074.703,E2 -8074.703} C_VEL
LIN {X 0,Y 460.503,Z 136.119,A -85,B 0,C 180,E1 -8077.571,E2 -8077.571} C_VEL
LIN {X 0,Y 460.561,Z 136.112,A -85,B 0,C 180,E1 -8080.384,E2 -8080.384} C_VEL
LIN {X 0,Y 460.567,Z 136.114,A -85,B 0,C 180,E1 -8084.058,E2 -8084.058} C_VEL
LIN {X 0,Y 460.601,Z 136.106,A -85,B 0,C 180,E1 -8087.666,E2 -8087.666} C_VEL
LIN {X 0,Y 460.583,Z 136.103,A -85,B 0,C 180,E1 -8091.223,E2 -8091.223} C_VEL
LIN {X 0,Y 460.664,Z 136.103,A -85,B 0,C 180,E1 -8093.87,E2 -8093.87} C_VEL
LIN {X 0,Y 460.752,Z 136.083,A -85,B 0,C 180,E1 -8097.377,E2 -8097.377} C_VEL
LIN {X 0,Y 460.817,Z 136.086,A -85,B 0,C 180,E1 -8100,E2 -8100} C_VEL
LIN {X 0,Y 460.755,Z 136.082,A -85,B 0,C 180,E1 -8102.623,E2 -8102.623} C_VEL
LIN {X 0,Y 460.666,Z 136.101,A -85,B 0,C 180,E1 -8106.131,E2 -8106.131} C_VEL
LIN {X 0,Y 460.614,Z 136.099,A -85,B 0,C 180,E1 -8108.777,E2 -8108.777} C_VEL
LIN {X 0,Y 460.597,Z 136.107,A -85,B 0,C 180,E1 -8112.435,E2 -8112.435} C_VEL
LIN {X 0,Y 460.602,Z 136.108,A -85,B 0,C 180,E1 -8115.998,E2 -8115.998} C_VEL
LIN {X 0,Y 460.568,Z 136.111,A -85,B 0,C 180,E1 -8119.616,E2 -8119.616} C_VEL
LIN {X 0,Y 460.508,Z 136.119,A -85,B 0,C 180,E1 -8122.429,E2 -8122.429} C_VEL
LIN {X 0,Y 460.548,Z 136.114,A -85,B 0,C 180,E1 -8125.797,E2 -8125.797} C_VEL
LIN {X 0,Y 460.528,Z 136.115,A -85,B 0,C 180,E1 -8128.235,E2 -8128.235} C_VEL
LIN {X 0,Y 460.521,Z 136.119,A -85,B 0,C 180,E1 -8131.283,E2 -8131.283} C_VEL
LIN {X 0,Y 460.525,Z 136.121,A -85,B 0,C 180,E1 -8134.504,E2 -8134.504} C_VEL
LIN {X 0,Y 460.503,Z 136.119,A -85,B 0,C 180,E1 -8137.623,E2 -8137.623} C_VEL
LIN {X 0,Y 460.541,Z 136.114,A -85,B 0,C 180,E1 -8140.269,E2 -8140.269} C_VEL
LIN {X 0,Y 460.501,Z 136.119,A -85,B 0,C 180,E1 -8143.376,E2 -8143.376} C_VEL
LIN {X 0,Y 460.511,Z 136.122,A -85,B 0,C 180,E1 -8146.626,E2 -8146.626} C_VEL
LIN {X 0,Y 460.54,Z 136.118,A -85,B 0,C 180,E1 -8149.731,E2 -8149.731} C_VEL
LIN {X 0,Y 460.503,Z 136.122,A -85,B 0,C 180,E1 -8152.524,E2 -8152.524} C_VEL
LIN {X 0,Y 460.55,Z 136.118,A -85,B 0,C 180,E1 -8155.624,E2 -8155.624} C_VEL
LIN {X 0,Y 460.542,Z 136.116,A -85,B 0,C 180,E1 -8158.744,E2 -8158.744} C_VEL
LIN {X 0,Y 460.585,Z 136.115,A -85,B 0,C 180,E1 -8162.254,E2 -8162.254} C_VEL
LIN {X 0,Y 460.601,Z 136.137,A -85,B 0,C 180,E1 -8164.506,E2 -8164.506} C_VEL
LIN {X 0,Y 461.76,Z 142.609,A -85,B 0,C 180,E1 -8165.952,E2 -8165.952} C_VEL
LIN {X 0,Y 461.748,Z 150.618,A -85,B 0,C 180,E1 -8167.634,E2 -8167.634} C_VEL
LIN {X 0,Y 464.91,Z 165.279,A -85,B 0,C 180,E1 -8168.023,E2 -8168.023} C_VEL
LIN {X 0,Y 464.348,Z 236.877,A -85,B 0,C 180,E1 -8169.142,E2 -8169.142} C_VEL
LIN {X 0,Y 463.667,Z 240.808,A -85,B 0,C 180,E1 -8169.177,E2 -8169.177} C_VEL
LIN {X 0,Y 457.964,Z 253.099,A -85,B 0,C 180,E1 -8169.152,E2 -8169.152} C_VEL
LIN {X 0,Y 457.389,Z 257.002,A -85,B 0,C 180,E1 -8169.204,E2 -8169.204} C_VEL
LIN {X 0,Y 457.035,Z 270.027,A -85,B 0,C 180,E1 -8169.569,E2 -8169.569} C_VEL
LIN {X 0,Y 456.635,Z 282.983,A -85,B 0,C 180,E1 -8170.127,E2 -8170.127} C_VEL
LIN {X 0,Y 456.223,Z 294.095,A -85,B 0,C 180,E1 -8170.775,E2 -8170.775} C_VEL
LIN {X 0,Y 455.634,Z 304.792,A -85,B 0,C 180,E1 -8171.566,E2 -8171.566} C_VEL
LIN {X 0,Y 455.05,Z 315.682,A -85,B 0,C 180,E1 -8172.588,E2 -8172.588} C_VEL
LIN {X 0,Y 454.588,Z 324.406,A -85,B 0,C 180,E1 -8173.593,E2 -8173.593} C_VEL
LIN {X 0,Y 454.078,Z 332.658,A -85,B 0,C 180,E1 -8174.744,E2 -8174.744} C_VEL
LIN {X 0,Y 453.579,Z 340.59,A -85,B 0,C 180,E1 -8176.103,E2 -8176.103} C_VEL
LIN {X 0,Y 453.212,Z 346.889,A -85,B 0,C 180,E1 -8177.461,E2 -8177.461} C_VEL
LIN {X 0,Y 452.944,Z 351.879,A -85,B 0,C 180,E1 -8178.816,E2 -8178.816} C_VEL
LIN {X 0,Y 452.707,Z 355.728,A -85,B 0,C 180,E1 -8180.167,E2 -8180.167} C_VEL
LIN {X 0,Y 452.662,Z 357.701,A -85,B 0,C 180,E1 -8181.067,E2 -8181.067} C_VEL
LIN {X 0,Y 452.604,Z 359.26,A -85,B 0,C 180,E1 -8181.966,E2 -8181.966} C_VEL
LIN {X 0,Y 452.632,Z 361.002,A -85,B 0,C 180,E1 -8183.581,E2 -8183.581} C_VEL
LIN {X 0,Y 452.578,Z 361.42,A -85,B 0,C 180,E1 -8184.653,E2 -8184.653} C_VEL
LIN {X 0,Y 452.499,Z 361.367,A -85,B 0,C 180,E1 -8185.545,E2 -8185.545} C_VEL
LIN {X 0,Y 452.608,Z 360.909,A -85,B 0,C 180,E1 -8186.438,E2 -8186.438} C_VEL
LIN {X 0,Y 452.555,Z 358.772,A -85,B 0,C 180,E1 -8188.219,E2 -8188.219} C_VEL
LIN {X 0,Y 452.586,Z 356.102,A -85,B 0,C 180,E1 -8189.554,E2 -8189.554} C_VEL
LIN {X 0,Y 452.67,Z 352.433,A -85,B 0,C 180,E1 -8190.889,E2 -8190.889} C_VEL
LIN {X 0,Y 453.011,Z 347.65,A -85,B 0,C 180,E1 -8192.222,E2 -8192.222} C_VEL
LIN {X 0,Y 453.187,Z 341.643,A -85,B 0,C 180,E1 -8193.556,E2 -8193.556} C_VEL
LIN {X 0,Y 453.681,Z 334.163,A -85,B 0,C 180,E1 -8194.887,E2 -8194.887} C_VEL
LIN {X 0,Y 454.16,Z 326.521,A -85,B 0,C 180,E1 -8195.995,E2 -8195.995} C_VEL
LIN {X 0,Y 454.68,Z 317.21,A -85,B 0,C 180,E1 -8197.102,E2 -8197.102} C_VEL
LIN {X 0,Y 455.249,Z 306.877,A -85,B 0,C 180,E1 -8198.097,E2 -8198.097} C_VEL
LIN {X 0,Y 455.798,Z 295.483,A -85,B 0,C 180,E1 -8198.975,E2 -8198.975} C_VEL
LIN {X 0,Y 456.16,Z 284.026,A -85,B 0,C 180,E1 -8199.663,E2 -8199.663} C_VEL
LIN {X 0,Y 456.472,Z 271.286,A -85,B 0,C 180,E1 -8200.225,E2 -8200.225} C_VEL
LIN {X 0,Y 456.787,Z 258.22,A -85,B 0,C 180,E1 -8200.61,E2 -8200.61} C_VEL
LIN {X 0,Y 457.504,Z 166.082,A -85,B 0,C 180,E1 -8202.08,E2 -8202.08} C_VEL
LIN {X 0,Y 454.496,Z 150.838,A -85,B 0,C 180,E1 -8202.445,E2 -8202.445} C_VEL
LIN {X 0,Y 454.574,Z 142.941,A -85,B 0,C 180,E1 -8204.092,E2 -8204.092} C_VEL
LIN {X 0,Y 453.599,Z 136.984,A -85,B 0,C 180,E1 -8205.429,E2 -8205.429} C_VEL
LIN {X 0,Y 453.518,Z 136.99,A -85,B 0,C 180,E1 -8209.038,E2 -8209.038} C_VEL
LIN {X 0,Y 453.477,Z 136.997,A -85,B 0,C 180,E1 -8211.835,E2 -8211.835} C_VEL
LIN {X 0,Y 453.5,Z 136.993,A -85,B 0,C 180,E1 -8214.734,E2 -8214.734} C_VEL
LIN {X 0,Y 453.53,Z 136.993,A -85,B 0,C 180,E1 -8217.958,E2 -8217.958} C_VEL
LIN {X 0,Y 453.463,Z 136.998,A -85,B 0,C 180,E1 -8221.524,E2 -8221.524} C_VEL
LIN {X 0,Y 453.484,Z 136.995,A -85,B 0,C 180,E1 -8224.776,E2 -8224.776} C_VEL
LIN {X 0,Y 453.46,Z 136.999,A -85,B 0,C 180,E1 -8228.31,E2 -8228.31} C_VEL
LIN {X 0,Y 453.489,Z 136.995,A -85,B 0,C 180,E1 -8230.608,E2 -8230.608} C_VEL
LIN {X 0,Y 453.449,Z 137.001,A -85,B 0,C 180,E1 -8233.243,E2 -8233.243} C_VEL
LIN {X 0,Y 453.455,Z 137.002,A -85,B 0,C 180,E1 -8235.777,E2 -8235.777} C_VEL
LIN {X 0,Y 453.472,Z 136.997,A -85,B 0,C 180,E1 -8238.208,E2 -8238.208} C_VEL
LIN {X 0,Y 453.479,Z 136.996,A -85,B 0,C 180,E1 -8240.793,E2 -8240.793} C_VEL
LIN {X 0,Y 453.445,Z 137.001,A -85,B 0,C 180,E1 -8243.916,E2 -8243.916} C_VEL
LIN {X 0,Y 453.47,Z 137,A -85,B 0,C 180,E1 -8247.15,E2 -8247.15} C_VEL
LIN {X 0,Y 453.464,Z 136.999,A -85,B 0,C 180,E1 -8250.267,E2 -8250.267} C_VEL
LIN {X 0,Y 453.522,Z 136.992,A -85,B 0,C 180,E1 -8252.296,E2 -8252.296} C_VEL
LIN {X 0,Y 453.481,Z 136.999,A -85,B 0,C 180,E1 -8255.263,E2 -8255.263} C_VEL
LIN {X 0,Y 453.469,Z 136.998,A -85,B 0,C 180,E1 -8258.414,E2 -8258.414} C_VEL
LIN {X 0,Y 453.511,Z 136.996,A -85,B 0,C 180,E1 -8261.008,E2 -8261.008} C_VEL
LIN {X 0,Y 453.526,Z 136.993,A -85,B 0,C 180,E1 -8263.893,E2 -8263.893} C_VEL
LIN {X 0,Y 453.552,Z 136.988,A -85,B 0,C 180,E1 -8267.471,E2 -8267.471} C_VEL
LIN {X 0,Y 453.57,Z 136.986,A -85,B 0,C 180,E1 -8271.086,E2 -8271.086} C_VEL
LIN {X 0,Y 453.624,Z 136.981,A -85,B 0,C 180,E1 -8273.774,E2 -8273.774} C_VEL
LIN {X 0,Y 453.69,Z 136.972,A -85,B 0,C 180,E1 -8277.336,E2 -8277.336} C_VEL
LIN {X 0,Y 453.754,Z 136.963,A -85,B 0,C 180,E1 -8280,E2 -8280} C_VEL
LIN {X 0,Y 453.691,Z 136.971,A -85,B 0,C 180,E1 -8282.664,E2 -8282.664} C_VEL
LIN {X 0,Y 453.628,Z 136.979,A -85,B 0,C 180,E1 -8286.226,E2 -8286.226} C_VEL
LIN {X 0,Y 453.57,Z 136.986,A -85,B 0,C 180,E1 -8288.914,E2 -8288.914} C_VEL
LIN {X 0,Y 453.552,Z 136.988,A -85,B 0,C 180,E1 -8292.529,E2 -8292.529} C_VEL
LIN {X 0,Y 453.532,Z 136.991,A -85,B 0,C 180,E1 -8296.196,E2 -8296.196} C_VEL
LIN {X 0,Y 453.505,Z 136.997,A -85,B 0,C 180,E1 -8299.04,E2 -8299.04} C_VEL
LIN {X 0,Y 453.464,Z 136.999,A -85,B 0,C 180,E1 -8301.837,E2 -8301.837} C_VEL
LIN {X 0,Y 453.48,Z 136.999,A -85,B 0,C 180,E1 -8304.736,E2 -8304.736} C_VEL
LIN {X 0,Y 453.518,Z 136.992,A -85,B 0,C 180,E1 -8307.959,E2 -8307.959} C_VEL
LIN {X 0,Y 453.455,Z 136.999,A -85,B 0,C 180,E1 -8311.526,E2 -8311.526} C_VEL
LIN {X 0,Y 453.473,Z 137,A -85,B 0,C 180,E1 -8314.777,E2 -8314.777} C_VEL
LIN {X 0,Y 453.452,Z 137.002,A -85,B 0,C 180,E1 -8318.313,E2 -8318.313} C_VEL
LIN {X 0,Y 453.486,Z 136.999,A -85,B 0,C 180,E1 -8320.61,E2 -8320.61} C_VEL
LIN {X 0,Y 453.445,Z 137,A -85,B 0,C 180,E1 -8323.245,E2 -8323.245} C_VEL
LIN {X 0,Y 453.457,Z 136.999,A -85,B 0,C 180,E1 -8325.78,E2 -8325.78} C_VEL
LIN {X 0,Y 453.473,Z 137.001,A -85,B 0,C 180,E1 -8328.21,E2 -8328.21} C_VEL
LIN {X 0,Y 453.51,Z 136.992,A -85,B 0,C 180,E1 -8330.791,E2 -8330.791} C_VEL
LIN {X 0,Y 453.449,Z 137.002,A -85,B 0,C 180,E1 -8333.918,E2 -8333.918} C_VEL
LIN {X 0,Y 453.479,Z 136.994,A -85,B 0,C 180,E1 -8337.152,E2 -8337.152} C_VEL
LIN {X 0,Y 453.472,Z 137.002,A -85,B 0,C 180,E1 -8340.27,E2 -8340.27} C_VEL
LIN {X 0,Y 453.57,Z 137.093,A -85,B 0,C 180,E1 -8343.345,E2 -8343.345} C_VEL
LIN {X 0,Y 455.847,Z 149.205,A -85,B 0,C 180,E1 -8345.617,E2 -8345.617} C_VEL
LIN {X 0,Y 455.181,Z 165.714,A -85,B 0,C 180,E1 -8348.489,E2 -8348.489} C_VEL
LIN {X 0,Y 454.38,Z 184.698,A -85,B 0,C 180,E1 -8351.748,E2 -8351.748} C_VEL
LIN {X 0,Y 454.217,Z 189.481,A -85,B 0,C 180,E1 -8352.565,E2 -8352.565} C_VEL
LIN {X 0,Y 457.296,Z 212.314,A -85,B 0,C 180,E1 -8353.046,E2 -8353.046} C_VEL
LIN {X 0,Y 456.644,Z 297.896,A -85,B 0,C 180,E1 -8354.405,E2 -8354.405} C_VEL
LIN {X 0,Y 456.177,Z 310.536,A -85,B 0,C 180,E1 -8354.761,E2 -8354.761} C_VEL
LIN {X 0,Y 455.721,Z 323.563,A -85,B 0,C 180,E1 -8355.317,E2 -8355.317} C_VEL
LIN {X 0,Y 455.128,Z 335.911,A -85,B 0,C 180,E1 -8356.039,E2 -8356.039} C_VEL
LIN {X 0,Y 454.576,Z 347.317,A -85,B 0,C 180,E1 -8356.911,E2 -8356.911} C_VEL
LIN {X 0,Y 453.995,Z 358.065,A -85,B 0,C 180,E1 -8357.938,E2 -8357.938} C_VEL
LIN {X 0,Y 453.594,Z 367.509,A -85,B 0,C 180,E1 -8359.06,E2 -8359.06} C_VEL
LIN {X 0,Y 453.127,Z 376.622,A -85,B 0,C 180,E1 -8360.403,E2 -8360.403} C_VEL
LIN {X 0,Y 452.831,Z 383.968,A -85,B 0,C 180,E1 -8361.747,E2 -8361.747} C_VEL
LIN {X 0,Y 452.667,Z 388.938,A -85,B 0,C 180,E1 -8362.866,E2 -8362.866} C_VEL
LIN {X 0,Y 452.543,Z 393.763,A -85,B 0,C 180,E1 -8364.207,E2 -8364.207} C_VEL
LIN {X 0,Y 452.486,Z 397.46,A -85,B 0,C 180,E1 -8365.547,E2 -8365.547} C_VEL
LIN {X 0,Y 452.521,Z 399.372,A -85,B 0,C 180,E1 -8366.439,E2 -8366.439} C_VEL
LIN {X 0,Y 452.53,Z 400.826,A -85,B 0,C 180,E1 -8367.33,E2 -8367.33} C_VEL
LIN {X 0,Y 452.494,Z 402.489,A -85,B 0,C 180,E1 -8369.111,E2 -8369.111} C_VEL
LIN {X 0,Y 452.475,Z 402.737,A -85,B 0,C 180,E1 -8370.001,E2 -8370.001} C_VEL
LIN {X 0,Y 452.494,Z 402.567,A -85,B 0,C 180,E1 -8370.891,E2 -8370.891} C_VEL
LIN {X 0,Y 452.527,Z 401.008,A -85,B 0,C 180,E1 -8372.671,E2 -8372.671} C_VEL
LIN {X 0,Y 452.492,Z 399.637,A -85,B 0,C 180,E1 -8373.563,E2 -8373.563} C_VEL
LIN {X 0,Y 452.541,Z 396.744,A -85,B 0,C 180,E1 -8374.901,E2 -8374.901} C_VEL
LIN {X 0,Y 452.554,Z 392.53,A -85,B 0,C 180,E1 -8376.332,E2 -8376.332} C_VEL
LIN {X 0,Y 452.733,Z 387.775,A -85,B 0,C 180,E1 -8377.583,E2 -8377.583} C_VEL
LIN {X 0,Y 452.984,Z 381.447,A -85,B 0,C 180,E1 -8378.926,E2 -8378.926} C_VEL
LIN {X 0,Y 453.362,Z 373.535,A -85,B 0,C 180,E1 -8380.27,E2 -8380.27} C_VEL
LIN {X 0,Y 454.002,Z 363.705,A -85,B 0,C 180,E1 -8381.61,E2 -8381.61} C_VEL
LIN {X 0,Y 454.449,Z 354.499,A -85,B 0,C 180,E1 -8382.631,E2 -8382.631} C_VEL
LIN {X 0,Y 455.07,Z 343.374,A -85,B 0,C 180,E1 -8383.623,E2 -8383.623} C_VEL
LIN {X 0,Y 455.654,Z 332.373,A -85,B 0,C 180,E1 -8384.402,E2 -8384.402} C_VEL
LIN {X 0,Y 456.24,Z 320.2,A -85,B 0,C 180,E1 -8385.067,E2 -8385.067} C_VEL
LIN {X 0,Y 456.74,Z 307.508,A -85,B 0,C 180,E1 -8385.565,E2 -8385.565} C_VEL
LIN {X 0,Y 457.177,Z 294.143,A -85,B 0,C 180,E1 -8385.893,E2 -8385.893} C_VEL
LIN {X 0,Y 457.737,Z 210.718,A -85,B 0,C 180,E1 -8387.224,E2 -8387.224} C_VEL
LIN {X 0,Y 454.414,Z 189.273,A -85,B 0,C 180,E1 -8387.731,E2 -8387.731} C_VEL
LIN {X 0,Y 455.1,Z 172.935,A -85,B 0,C 180,E1 -8390.569,E2 -8390.569} C_VEL
LIN {X 0,Y 456.063,Z 155.561,A -85,B 0,C 180,E1 -8393.62,E2 -8393.62} C_VEL
LIN {X 0,Y 456.138,Z 149.975,A -85,B 0,C 180,E1 -8394.625,E2 -8394.625} C_VEL
LIN {X 0,Y 453.76,Z 138.098,A -85,B 0,C 180,E1 -8396.939,E2 -8396.939} C_VEL
LIN {X 0,Y 453.514,Z 136.995,A -85,B 0,C 180,E1 -8397.204,E2 -8397.204} C_VEL
LIN {X 0,Y 453.471,Z 137.005,A -85,B 0,C 180,E1 -8399.784,E2 -8399.784} C_VEL
LIN {X 0,Y 453.493,Z 136.997,A -85,B 0,C 180,E1 -8403.189,E2 -8403.189} C_VEL
LIN {X 0,Y 453.453,Z 136.998,A -85,B 0,C 180,E1 -8406.299,E2 -8406.299} C_VEL
LIN {X 0,Y 453.466,Z 136.998,A -85,B 0,C 180,E1 -8409.453,E2 -8409.453} C_VEL
LIN {X 0,Y 453.461,Z 136.999,A -85,B 0,C 180,E1 -8411.932,E2 -8411.932} C_VEL
LIN {X 0,Y 453.484,Z 137,A -85,B 0,C 180,E1 -8415.472,E2 -8415.472} C_VEL
LIN {X 0,Y 453.461,Z 136.997,A -85,B 0,C 180,E1 -8418.207,E2 -8418.207} C_VEL
LIN {X 0,Y 453.449,Z 137.001,A -85,B 0,C 180,E1 -8420.801,E2 -8420.801} C_VEL
LIN {X 0,Y 453.454,Z 136.999,A -85,B 0,C 180,E1 -8423.917,E2 -8423.917} C_VEL
LIN {X 0,Y 453.478,Z 137,A -85,B 0,C 180,E1 -8427.151,E2 -8427.151} C_VEL
LIN {X 0,Y 453.461,Z 136.997,A -85,B 0,C 180,E1 -8430.267,E2 -8430.267} C_VEL
LIN {X 0,Y 453.455,Z 136.999,A -85,B 0,C 180,E1 -8433.291,E2 -8433.291} C_VEL
LIN {X 0,Y 453.492,Z 136.995,A -85,B 0,C 180,E1 -8436.238,E2 -8436.238} C_VEL
LIN {X 0,Y 453.474,Z 136.994,A -85,B 0,C 180,E1 -8439.117,E2 -8439.117} C_VEL
LIN {X 0,Y 453.484,Z 136.992,A -85,B 0,C 180,E1 -8441.943,E2 -8441.943} C_VEL
LIN {X 0,Y 453.516,Z 136.988,A -85,B 0,C 180,E1 -8444.726,E2 -8444.726} C_VEL
LIN {X 0,Y 453.564,Z 136.982,A -85,B 0,C 180,E1 -8447.471,E2 -8447.471} C_VEL
LIN {X 0,Y 453.553,Z 136.979,A -85,B 0,C 180,E1 -8451.086,E2 -8451.086} C_VEL
LIN {X 0,Y 453.633,Z 136.977,A -85,B 0,C 180,E1 -8453.774,E2 -8453.774} C_VEL
LIN {X 0,Y 453.699,Z 136.962,A -85,B 0,C 180,E1 -8457.337,E2 -8457.337} C_VEL
LIN {X 0,Y 453.766,Z 136.964,A -85,B 0,C 180,E1 -8460,E2 -8460} C_VEL
LIN {X 0,Y 453.702,Z 136.96,A -85,B 0,C 180,E1 -8462.664,E2 -8462.664} C_VEL
LIN {X 0,Y 453.634,Z 136.976,A -85,B 0,C 180,E1 -8466.226,E2 -8466.226} C_VEL
LIN {X 0,Y 453.581,Z 136.976,A -85,B 0,C 180,E1 -8468.914,E2 -8468.914} C_VEL
LIN {X 0,Y 453.565,Z 136.983,A -85,B 0,C 180,E1 -8472.529,E2 -8472.529} C_VEL
LIN {X 0,Y 453.545,Z 136.986,A -85,B 0,C 180,E1 -8476.196,E2 -8476.196} C_VEL
LIN {X 0,Y 453.518,Z 136.992,A -85,B 0,C 180,E1 -8479.039,E2 -8479.039} C_VEL
LIN {X 0,Y 453.476,Z 136.995,A -85,B 0,C 180,E1 -8481.836,E2 -8481.836} C_VEL
LIN {X 0,Y 453.494,Z 136.992,A -85,B 0,C 180,E1 -8484.736,E2 -8484.736} C_VEL
LIN {X 0,Y 453.508,Z 136.989,A -85,B 0,C 180,E1 -8487.953,E2 -8487.953} C_VEL
LIN {X 0,Y 453.477,Z 137,A -85,B 0,C 180,E1 -8490.76,E2 -8490.76} C_VEL
LIN {X 0,Y 453.47,Z 136.995,A -85,B 0,C 180,E1 -8493.914,E2 -8493.914} C_VEL
LIN {X 0,Y 453.454,Z 136.998,A -85,B 0,C 180,E1 -8497.19,E2 -8497.19} C_VEL
LIN {X 0,Y 453.496,Z 136.986,A -85,B 0,C 180,E1 -8500.609,E2 -8500.609} C_VEL
LIN {X 0,Y 453.457,Z 136.997,A -85,B 0,C 180,E1 -8503.244,E2 -8503.244} C_VEL
LIN {X 0,Y 453.463,Z 136.997,A -85,B 0,C 180,E1 -8505.778,E2 -8505.778} C_VEL
LIN {X 0,Y 453.497,Z 136.993,A -85,B 0,C 180,E1 -8509.409,E2 -8509.409} C_VEL
LIN {X 0,Y 453.456,Z 136.998,A -85,B 0,C 180,E1 -8512.81,E2 -8512.81} C_VEL
LIN {X 0,Y 453.481,Z 137,A -85,B 0,C 180,E1 -8516.087,E2 -8516.087} C_VEL
LIN {X 0,Y 453.481,Z 136.996,A -85,B 0,C 180,E1 -8519.24,E2 -8519.24} C_VEL
LIN {X 0,Y 453.54,Z 136.993,A -85,B 0,C 180,E1 -8522.297,E2 -8522.297} C_VEL
LIN {X 0,Y 453.555,Z 137.029,A -85,B 0,C 180,E1 -8524.286,E2 -8524.286} C_VEL
LIN {X 0,Y 454.899,Z 144.796,A -85,B 0,C 180,E1 -8526.038,E2 -8526.038} C_VEL
LIN {X 0,Y 454.829,Z 151.028,A -85,B 0,C 180,E1 -8527.355,E2 -8527.355} C_VEL
LIN {X 0,Y 458.208,Z 166.924,A -85,B 0,C 180,E1 -8527.764,E2 -8527.764} C_VEL
LIN {X 0,Y 457.389,Z 257.002,A -85,B 0,C 180,E1 -8529.204,E2 -8529.204} C_VEL
LIN {X 0,Y 456.884,Z 262.791,A -85,B 0,C 180,E1 -8529.322,E2 -8529.322} C_VEL
LIN {X 0,Y 454.006,Z 272.132,A -85,B 0,C 180,E1 -8529.515,E2 -8529.515} C_VEL
LIN {X 0,Y 450.773,Z 281.254,A -85,B 0,C 180,E1 -8529.797,E2 -8529.797} C_VEL
LIN {X 0,Y 449.725,Z 286.709,A -85,B 0,C 180,E1 -8530.056,E2 -8530.056} C_VEL
LIN {X 0,Y 449.166,Z 298.514,A -85,B 0,C 180,E1 -8530.817,E2 -8530.817} C_VEL
LIN {X 0,Y 448.488,Z 309.679,A -85,B 0,C 180,E1 -8531.735,E2 -8531.735} C_VEL
LIN {X 0,Y 447.868,Z 320.486,A -85,B 0,C 180,E1 -8532.867,E2 -8532.867} C_VEL
LIN {X 0,Y 447.392,Z 329.537,A -85,B 0,C 180,E1 -8534.043,E2 -8534.043} C_VEL
LIN {X 0,Y 446.844,Z 336.835,A -85,B 0,C 180,E1 -8535.191,E2 -8535.191} C_VEL
LIN {X 0,Y 446.367,Z 343.989,A -85,B 0,C 180,E1 -8536.571,E2 -8536.571} C_VEL
LIN {X 0,Y 446.117,Z 349.065,A -85,B 0,C 180,E1 -8537.789,E2 -8537.789} C_VEL
LIN {X 0,Y 445.823,Z 353.447,A -85,B 0,C 180,E1 -8539.095,E2 -8539.095} C_VEL
LIN {X 0,Y 445.652,Z 355.92,A -85,B 0,C 180,E1 -8540.01,E2 -8540.01} C_VEL
LIN {X 0,Y 445.581,Z 357.915,A -85,B 0,C 180,E1 -8540.924,E2 -8540.924} C_VEL
LIN {X 0,Y 445.527,Z 359.494,A -85,B 0,C 180,E1 -8541.837,E2 -8541.837} C_VEL
LIN {X 0,Y 445.552,Z 360.662,A -85,B 0,C 180,E1 -8542.75,E2 -8542.75} C_VEL
LIN {X 0,Y 445.532,Z 361.391,A -85,B 0,C 180,E1 -8543.66,E2 -8543.66} C_VEL
LIN {X 0,Y 445.493,Z 361.734,A -85,B 0,C 180,E1 -8544.568,E2 -8544.568} C_VEL
LIN {X 0,Y 445.504,Z 361.276,A -85,B 0,C 180,E1 -8546.381,E2 -8546.381} C_VEL
LIN {X 0,Y 445.502,Z 360.426,A -85,B 0,C 180,E1 -8547.287,E2 -8547.287} C_VEL
LIN {X 0,Y 445.477,Z 357.549,A -85,B 0,C 180,E1 -8549.095,E2 -8549.095} C_VEL
LIN {X 0,Y 445.644,Z 354.255,A -85,B 0,C 180,E1 -8550.451,E2 -8550.451} C_VEL
LIN {X 0,Y 445.734,Z 349.916,A -85,B 0,C 180,E1 -8551.806,E2 -8551.806} C_VEL
LIN {X 0,Y 446.091,Z 344.387,A -85,B 0,C 180,E1 -8553.16,E2 -8553.16} C_VEL
LIN {X 0,Y 446.45,Z 337.497,A -85,B 0,C 180,E1 -8554.514,E2 -8554.514} C_VEL
LIN {X 0,Y 447.063,Z 328.853,A -85,B 0,C 180,E1 -8555.864,E2 -8555.864} C_VEL
LIN {X 0,Y 447.564,Z 320.021,A -85,B 0,C 180,E1 -8556.989,E2 -8556.989} C_VEL
LIN {X 0,Y 448.167,Z 310.307,A -85,B 0,C 180,E1 -8557.999,E2 -8557.999} C_VEL
LIN {X 0,Y 448.664,Z 299.629,A -85,B 0,C 180,E1 -8558.898,E2 -8558.898} C_VEL
LIN {X 0,Y 449.119,Z 288.283,A -85,B 0,C 180,E1 -8559.648,E2 -8559.648} C_VEL
LIN {X 0,Y 449.533,Z 275.175,A -85,B 0,C 180,E1 -8560.3,E2 -8560.3} C_VEL
LIN {X 0,Y 449.841,Z 263,A -85,B 0,C 180,E1 -8560.719,E2 -8560.719} C_VEL
LIN {X 0,Y 449.98,Z 247.603,A -85,B 0,C 180,E1 -8561.029,E2 -8561.029} C_VEL
LIN {X 0,Y 450.723,Z 167.187,A -85,B 0,C 180,E1 -8562.307,E2 -8562.307} C_VEL
LIN {X 0,Y 447.515,Z 151.128,A -85,B 0,C 180,E1 -8562.7,E2 -8562.7} C_VEL
LIN {X 0,Y 447.528,Z 143.481,A -85,B 0,C 180,E1 -8564.319,E2 -8564.319} C_VEL
LIN {X 0,Y 446.545,Z 137.864,A -85,B 0,C 180,E1 -8565.608,E2 -8565.608} C_VEL
LIN {X 0,Y 446.469,Z 137.867,A -85,B 0,C 180,E1 -8569.302,E2 -8569.302} C_VEL
LIN {X 0,Y 446.419,Z 137.88,A -85,B 0,C 180,E1 -8572.198,E2 -8572.198} C_VEL
LIN {X 0,Y 446.443,Z 137.871,A -85,B 0,C 180,E1 -8575.152,E2 -8575.152} C_VEL
LIN {X 0,Y 446.483,Z 137.872,A -85,B 0,C 180,E1 -8578.177,E2 -8578.177} C_VEL
LIN {X 0,Y 446.417,Z 137.878,A -85,B 0,C 180,E1 -8581.774,E2 -8581.774} C_VEL
LIN {X 0,Y 446.426,Z 137.875,A -85,B 0,C 180,E1 -8584.522,E2 -8584.522} C_VEL
LIN {X 0,Y 446.412,Z 137.879,A -85,B 0,C 180,E1 -8588.078,E2 -8588.078} C_VEL
LIN {X 0,Y 446.422,Z 137.875,A -85,B 0,C 180,E1 -8590.916,E2 -8590.916} C_VEL
LIN {X 0,Y 446.394,Z 137.882,A -85,B 0,C 180,E1 -8593.845,E2 -8593.845} C_VEL
LIN {X 0,Y 446.39,Z 137.879,A -85,B 0,C 180,E1 -8596.403,E2 -8596.403} C_VEL
LIN {X 0,Y 446.42,Z 137.876,A -85,B 0,C 180,E1 -8599.081,E2 -8599.081} C_VEL
LIN {X 0,Y 446.399,Z 137.879,A -85,B 0,C 180,E1 -8602.12,E2 -8602.12} C_VEL
LIN {X 0,Y 446.414,Z 137.88,A -85,B 0,C 180,E1 -8605.475,E2 -8605.475} C_VEL
LIN {X 0,Y 446.406,Z 137.878,A -85,B 0,C 180,E1 -8608.699,E2 -8608.699} C_VEL
LIN {X 0,Y 446.475,Z 137.87,A -85,B 0,C 180,E1 -8611.82,E2 -8611.82} C_VEL
LIN {X 0,Y 446.426,Z 137.876,A -85,B 0,C 180,E1 -8614.846,E2 -8614.846} C_VEL
LIN {X 0,Y 446.437,Z 137.875,A -85,B 0,C 180,E1 -8618.245,E2 -8618.245} C_VEL
LIN {X 0,Y 446.435,Z 137.875,A -85,B 0,C 180,E1 -8621.648,E2 -8621.648} C_VEL
LIN {X 0,Y 446.465,Z 137.871,A -85,B 0,C 180,E1 -8624.478,E2 -8624.478} C_VEL
LIN {X 0,Y 446.504,Z 137.866,A -85,B 0,C 180,E1 -8628.193,E2 -8628.193} C_VEL
LIN {X 0,Y 446.518,Z 137.866,A -85,B 0,C 180,E1 -8630.944,E2 -8630.944} C_VEL
LIN {X 0,Y 446.594,Z 137.857,A -85,B 0,C 180,E1 -8633.675,E2 -8633.675} C_VEL
LIN {X 0,Y 446.639,Z 137.85,A -85,B 0,C 180,E1 -8637.294,E2 -8637.294} C_VEL
LIN {X 0,Y 446.705,Z 137.841,A -85,B 0,C 180,E1 -8640,E2 -8640} C_VEL
LIN {X 0,Y 446.64,Z 137.85,A -85,B 0,C 180,E1 -8642.706,E2 -8642.706} C_VEL
LIN {X 0,Y 446.597,Z 137.856,A -85,B 0,C 180,E1 -8646.324,E2 -8646.324} C_VEL
LIN {X 0,Y 446.518,Z 137.866,A -85,B 0,C 180,E1 -8649.056,E2 -8649.056} C_VEL
LIN {X 0,Y 446.509,Z 137.866,A -85,B 0,C 180,E1 -8652.73,E2 -8652.73} C_VEL
LIN {X 0,Y 446.476,Z 137.869,A -85,B 0,C 180,E1 -8656.46,E2 -8656.46} C_VEL
LIN {X 0,Y 446.456,Z 137.873,A -85,B 0,C 180,E1 -8659.304,E2 -8659.304} C_VEL
LIN {X 0,Y 446.405,Z 137.878,A -85,B 0,C 180,E1 -8662.2,E2 -8662.2} C_VEL
LIN {X 0,Y 446.425,Z 137.877,A -85,B 0,C 180,E1 -8665.154,E2 -8665.154} C_VEL
LIN {X 0,Y 446.475,Z 137.869,A -85,B 0,C 180,E1 -8668.179,E2 -8668.179} C_VEL
LIN {X 0,Y 446.408,Z 137.877,A -85,B 0,C 180,E1 -8671.775,E2 -8671.775} C_VEL
LIN {X 0,Y 446.414,Z 137.88,A -85,B 0,C 180,E1 -8674.524,E2 -8674.524} C_VEL
LIN {X 0,Y 446.404,Z 137.878,A -85,B 0,C 180,E1 -8678.08,E2 -8678.08} C_VEL
LIN {X 0,Y 446.419,Z 137.876,A -85,B 0,C 180,E1 -8680.919,E2 -8680.919} C_VEL
LIN {X 0,Y 446.391,Z 137.879,A -85,B 0,C 180,E1 -8683.847,E2 -8683.847} C_VEL
LIN {X 0,Y 446.391,Z 137.883,A -85,B 0,C 180,E1 -8686.405,E2 -8686.405} C_VEL
LIN {X 0,Y 446.421,Z 137.874,A -85,B 0,C 180,E1 -8689.084,E2 -8689.084} C_VEL
LIN {X 0,Y 446.41,Z 137.879,A -85,B 0,C 180,E1 -8691.922,E2 -8691.922} C_VEL
LIN {X 0,Y 446.424,Z 137.874,A -85,B 0,C 180,E1 -8695.478,E2 -8695.478} C_VEL
LIN {X 0,Y 446.412,Z 137.878,A -85,B 0,C 180,E1 -8698.701,E2 -8698.701} C_VEL
LIN {X 0,Y 446.482,Z 137.873,A -85,B 0,C 180,E1 -8701.823,E2 -8701.823} C_VEL
LIN {X 0,Y 446.52,Z 137.894,A -85,B 0,C 180,E1 -8703.13,E2 -8703.13} C_VEL
LIN {X 0,Y 448.706,Z 149.192,A -85,B 0,C 180,E1 -8705.291,E2 -8705.291} C_VEL
LIN {X 0,Y 448.884,Z 152.979,A -85,B 0,C 180,E1 -8705.98,E2 -8705.98} C_VEL
LIN {X 0,Y 447.967,Z 170.669,A -85,B 0,C 180,E1 -8709.09,E2 -8709.09} C_VEL
LIN {X 0,Y 447.223,Z 188.549,A -85,B 0,C 180,E1 -8712.204,E2 -8712.204} C_VEL
LIN {X 0,Y 447.205,Z 189.157,A -85,B 0,C 180,E1 -8712.309,E2 -8712.309} C_VEL
LIN {X 0,Y 450.454,Z 213.931,A -85,B 0,C 180,E1 -8712.836,E2 -8712.836} C_VEL
LIN {X 0,Y 449.775,Z 297.793,A -85,B 0,C 180,E1 -8714.19,E2 -8714.19} C_VEL
LIN {X 0,Y 449.26,Z 311.121,A -85,B 0,C 180,E1 -8714.578,E2 -8714.578} C_VEL
LIN {X 0,Y 448.764,Z 323.913,A -85,B 0,C 180,E1 -8715.142,E2 -8715.142} C_VEL
LIN {X 0,Y 448.221,Z 335.266,A -85,B 0,C 180,E1 -8715.819,E2 -8715.819} C_VEL
LIN {X 0,Y 447.601,Z 347.026,A -85,B 0,C 180,E1 -8716.729,E2 -8716.729} C_VEL
LIN {X 0,Y 447.022,Z 357.527,A -85,B 0,C 180,E1 -8717.747,E2 -8717.747} C_VEL
LIN {X 0,Y 446.595,Z 367.023,A -85,B 0,C 180,E1 -8718.886,E2 -8718.886} C_VEL
LIN {X 0,Y 446.086,Z 376.165,A -85,B 0,C 180,E1 -8720.25,E2 -8720.25} C_VEL
LIN {X 0,Y 445.772,Z 383.535,A -85,B 0,C 180,E1 -8721.615,E2 -8721.615} C_VEL
LIN {X 0,Y 445.595,Z 388.527,A -85,B 0,C 180,E1 -8722.752,E2 -8722.752} C_VEL
LIN {X 0,Y 445.451,Z 392.936,A -85,B 0,C 180,E1 -8723.978,E2 -8723.978} C_VEL
LIN {X 0,Y 445.412,Z 397.086,A -85,B 0,C 180,E1 -8725.476,E2 -8725.476} C_VEL
LIN {X 0,Y 445.419,Z 399.006,A -85,B 0,C 180,E1 -8726.382,E2 -8726.382} C_VEL
LIN {X 0,Y 445.455,Z 400.477,A -85,B 0,C 180,E1 -8727.288,E2 -8727.288} C_VEL
LIN {X 0,Y 445.4,Z 402.154,A -85,B 0,C 180,E1 -8729.097,E2 -8729.097} C_VEL
LIN {X 0,Y 445.41,Z 402.41,A -85,B 0,C 180,E1 -8730.001,E2 -8730.001} C_VEL
LIN {X 0,Y 445.401,Z 402.254,A -85,B 0,C 180,E1 -8730.905,E2 -8730.905} C_VEL
LIN {X 0,Y 445.451,Z 400.711,A -85,B 0,C 180,E1 -8732.714,E2 -8732.714} C_VEL
LIN {X 0,Y 445.391,Z 399.346,A -85,B 0,C 180,E1 -8733.62,E2 -8733.62} C_VEL
LIN {X 0,Y 445.468,Z 396.47,A -85,B 0,C 180,E1 -8734.979,E2 -8734.979} C_VEL
LIN {X 0,Y 445.456,Z 392.563,A -85,B 0,C 180,E1 -8736.341,E2 -8736.341} C_VEL
LIN {X 0,Y 445.68,Z 387.537,A -85,B 0,C 180,E1 -8737.704,E2 -8737.704} C_VEL
LIN {X 0,Y 445.943,Z 381.233,A -85,B 0,C 180,E1 -8739.068,E2 -8739.068} C_VEL
LIN {X 0,Y 446.331,Z 373.355,A -85,B 0,C 180,E1 -8740.433,E2 -8740.433} C_VEL
LIN {X 0,Y 446.929,Z 365.344,A -85,B 0,C 180,E1 -8741.567,E2 -8741.567} C_VEL
LIN {X 0,Y 447.412,Z 355.583,A -85,B 0,C 180,E1 -8742.705,E2 -8742.705} C_VEL
LIN {X 0,Y 448.063,Z 344.746,A -85,B 0,C 180,E1 -8743.724,E2 -8743.724} C_VEL
LIN {X 0,Y 448.686,Z 334.176,A -85,B 0,C 180,E1 -8744.515,E2 -8744.515} C_VEL
LIN {X 0,Y 449.326,Z 321.47,A -85,B 0,C 180,E1 -8745.247,E2 -8745.247} C_VEL
LIN {X 0,Y 449.943,Z 308.757,A -85,B 0,C 180,E1 -8745.777,E2 -8745.777} C_VEL
LIN {X 0,Y 450.37,Z 296.564,A -85,B 0,C 180,E1 -8746.11,E2 -8746.11} C_VEL
LIN {X 0,Y 451.039,Z 211.643,A -85,B 0,C 180,E1 -8747.493,E2 -8747.493} C_VEL
LIN {X 0,Y 447.473,Z 188.935,A -85,B 0,C 180,E1 -8748.042,E2 -8748.042} C_VEL
LIN {X 0,Y 448.305,Z 171.424,A -85,B 0,C 180,E1 -8751.136,E2 -8751.136} C_VEL
LIN {X 0,Y 449.318,Z 154.2,A -85,B 0,C 180,E1 -8754.216,E2 -8754.216} C_VEL
LIN {X 0,Y 449.015,Z 150.037,A -85,B 0,C 180,E1 -8755,E2 -8755} C_VEL
LIN {X 0,Y 446.478,Z 137.873,A -85,B 0,C 180,E1 -8757.447,E2 -8757.447} C_VEL
LIN {X 0,Y 446.428,Z 137.882,A -85,B 0,C 180,E1 -8760.25,E2 -8760.25} C_VEL
LIN {X 0,Y 446.448,Z 137.876,A -85,B 0,C 180,E1 -8763.454,E2 -8763.454} C_VEL
LIN {X 0,Y 446.402,Z 137.875,A -85,B 0,C 180,E1 -8766.746,E2 -8766.746} C_VEL
LIN {X 0,Y 446.438,Z 137.872,A -85,B 0,C 180,E1 -8770.199,E2 -8770.199} C_VEL
LIN {X 0,Y 446.4,Z 137.881,A -85,B 0,C 180,E1 -8773.597,E2 -8773.597} C_VEL
LIN {X 0,Y 446.399,Z 137.877,A -85,B 0,C 180,E1 -8776.404,E2 -8776.404} C_VEL
LIN {X 0,Y 446.406,Z 137.881,A -85,B 0,C 180,E1 -8779.086,E2 -8779.086} C_VEL
LIN {X 0,Y 446.407,Z 137.876,A -85,B 0,C 180,E1 -8782.121,E2 -8782.121} C_VEL
LIN {X 0,Y 446.423,Z 137.877,A -85,B 0,C 180,E1 -8785.476,E2 -8785.476} C_VEL
LIN {X 0,Y 446.415,Z 137.879,A -85,B 0,C 180,E1 -8788.7,E2 -8788.7} C_VEL
LIN {X 0,Y 446.426,Z 137.872,A -85,B 0,C 180,E1 -8791.836,E2 -8791.836} C_VEL
LIN {X 0,Y 446.421,Z 137.88,A -85,B 0,C 180,E1 -8794.845,E2 -8794.845} C_VEL
LIN {X 0,Y 446.447,Z 137.873,A -85,B 0,C 180,E1 -8798.246,E2 -8798.246} C_VEL
LIN {X 0,Y 446.439,Z 137.869,A -85,B 0,C 180,E1 -8801.648,E2 -8801.648} C_VEL
LIN {X 0,Y 446.457,Z 137.871,A -85,B 0,C 180,E1 -8804.478,E2 -8804.478} C_VEL
LIN {X 0,Y 446.516,Z 137.86,A -85,B 0,C 180,E1 -8807.384,E2 -8807.384} C_VEL
LIN {X 0,Y 446.504,Z 137.857,A -85,B 0,C 180,E1 -8810.944,E2 -8810.944} C_VEL
LIN {X 0,Y 446.603,Z 137.852,A -85,B 0,C 180,E1 -8813.676,E2 -8813.676} C_VEL
LIN {X 0,Y 446.648,Z 137.839,A -85,B 0,C 180,E1 -8817.294,E2 -8817.294} C_VEL
LIN {X 0,Y 446.716,Z 137.843,A -85,B 0,C 180,E1 -8820,E2 -8820} C_VEL
LIN {X 0,Y 446.651,Z 137.838,A -85,B 0,C 180,E1 -8822.706,E2 -8822.706} C_VEL
LIN {X 0,Y 446.604,Z 137.851,A -85,B 0,C 180,E1 -8826.324,E2 -8826.324} C_VEL
LIN {X 0,Y 446.529,Z 137.855,A -85,B 0,C 180,E1 -8829.056,E2 -8829.056} C_VEL
LIN {X 0,Y 446.522,Z 137.861,A -85,B 0,C 180,E1 -8832.73,E2 -8832.73} C_VEL
LIN {X 0,Y 446.489,Z 137.865,A -85,B 0,C 180,E1 -8836.459,E2 -8836.459} C_VEL
LIN {X 0,Y 446.469,Z 137.868,A -85,B 0,C 180,E1 -8839.303,E2 -8839.303} C_VEL
LIN {X 0,Y 446.417,Z 137.874,A -85,B 0,C 180,E1 -8842.2,E2 -8842.2} C_VEL
LIN {X 0,Y 446.439,Z 137.874,A -85,B 0,C 180,E1 -8845.154,E2 -8845.154} C_VEL
LIN {X 0,Y 446.45,Z 137.869,A -85,B 0,C 180,E1 -8848.181,E2 -8848.181} C_VEL
LIN {X 0,Y 446.416,Z 137.875,A -85,B 0,C 180,E1 -8851.301,E2 -8851.301} C_VEL
LIN {X 0,Y 446.425,Z 137.877,A -85,B 0,C 180,E1 -8854.524,E2 -8854.524} C_VEL
LIN {X 0,Y 446.415,Z 137.876,A -85,B 0,C 180,E1 -8858.079,E2 -8858.079} C_VEL
LIN {X 0,Y 446.431,Z 137.863,A -85,B 0,C 180,E1 -8861.391,E2 -8861.391} C_VEL
LIN {X 0,Y 446.454,Z 137.87,A -85,B 0,C 180,E1 -8864.896,E2 -8864.896} C_VEL
LIN {X 0,Y 446.422,Z 137.877,A -85,B 0,C 180,E1 -8868.608,E2 -8868.608} C_VEL
LIN {X 0,Y 446.429,Z 137.873,A -85,B 0,C 180,E1 -8870.971,E2 -8870.971} C_VEL
LIN {X 0,Y 446.423,Z 137.878,A -85,B 0,C 180,E1 -8874.374,E2 -8874.374} C_VEL
LIN {X 0,Y 446.426,Z 137.878,A -85,B 0,C 180,E1 -8877.638,E2 -8877.638} C_VEL
LIN {X 0,Y 446.452,Z 137.873,A -85,B 0,C 180,E1 -8880.79,E2 -8880.79} C_VEL
LIN {X 0,Y 446.533,Z 137.985,A -85,B 0,C 180,E1 -8884.071,E2 -8884.071} C_VEL
LIN {X 0,Y 447.962,Z 146.099,A -85,B 0,C 180,E1 -8885.926,E2 -8885.926} C_VEL
LIN {X 0,Y 447.934,Z 151.267,A -85,B 0,C 180,E1 -8887.034,E2 -8887.034} C_VEL
LIN {X 0,Y 451.44,Z 167.087,A -85,B 0,C 180,E1 -8887.469,E2 -8887.469} C_VEL
LIN {X 0,Y 450.601,Z 259.11,A -85,B 0,C 180,E1 -8888.977,E2 -8888.977} C_VEL
LIN {X 0,Y 450.212,Z 272.328,A -85,B 0,C 180,E1 -8889.38,E2 -8889.38} C_VEL
LIN {X 0,Y 449.79,Z 284.907,A -85,B 0,C 180,E1 -8889.953,E2 -8889.953} C_VEL
LIN {X 0,Y 449.725,Z 286.709,A -85,B 0,C 180,E1 -8890.056,E2 -8890.056} C_VEL
LIN {X 0,Y 448.717,Z 292.181,A -85,B 0,C 180,E1 -8890.351,E2 -8890.351} C_VEL
LIN {X 0,Y 445.524,Z 300.794,A -85,B 0,C 180,E1 -8890.845,E2 -8890.845} C_VEL
LIN {X 0,Y 442.389,Z 308.924,A -85,B 0,C 180,E1 -8891.428,E2 -8891.428} C_VEL
LIN {X 0,Y 441.457,Z 313.606,A -85,B 0,C 180,E1 -8891.856,E2 -8891.856} C_VEL
LIN {X 0,Y 440.9,Z 322.538,A -85,B 0,C 180,E1 -8892.856,E2 -8892.856} C_VEL
LIN {X 0,Y 440.365,Z 331.083,A -85,B 0,C 180,E1 -8894.019,E2 -8894.019} C_VEL
LIN {X 0,Y 439.727,Z 339.407,A -85,B 0,C 180,E1 -8895.42,E2 -8895.42} C_VEL
LIN {X 0,Y 439.26,Z 346.088,A -85,B 0,C 180,E1 -8896.82,E2 -8896.82} C_VEL
LIN {X 0,Y 438.884,Z 352.177,A -85,B 0,C 180,E1 -8898.453,E2 -8898.453} C_VEL
LIN {X 0,Y 438.599,Z 356.115,A -85,B 0,C 180,E1 -8899.847,E2 -8899.847} C_VEL
LIN {X 0,Y 438.512,Z 358.131,A -85,B 0,C 180,E1 -8900.777,E2 -8900.777} C_VEL
LIN {X 0,Y 438.468,Z 360.925,A -85,B 0,C 180,E1 -8902.632,E2 -8902.632} C_VEL
LIN {X 0,Y 438.47,Z 361.708,A -85,B 0,C 180,E1 -8903.601,E2 -8903.601} C_VEL
LIN {X 0,Y 438.343,Z 362.034,A -85,B 0,C 180,E1 -8905.401,E2 -8905.401} C_VEL
LIN {X 0,Y 438.402,Z 361.634,A -85,B 0,C 180,E1 -8906.323,E2 -8906.323} C_VEL
LIN {X 0,Y 438.427,Z 360.817,A -85,B 0,C 180,E1 -8907.243,E2 -8907.243} C_VEL
LIN {X 0,Y 438.413,Z 357.98,A -85,B 0,C 180,E1 -8909.081,E2 -8909.081} C_VEL
LIN {X 0,Y 438.56,Z 354.729,A -85,B 0,C 180,E1 -8910.458,E2 -8910.458} C_VEL
LIN {X 0,Y 438.669,Z 350.434,A -85,B 0,C 180,E1 -8911.835,E2 -8911.835} C_VEL
LIN {X 0,Y 439.032,Z 344.954,A -85,B 0,C 180,E1 -8913.211,E2 -8913.211} C_VEL
LIN {X 0,Y 439.424,Z 338.128,A -85,B 0,C 180,E1 -8914.586,E2 -8914.586} C_VEL
LIN {X 0,Y 440.058,Z 329.566,A -85,B 0,C 180,E1 -8915.958,E2 -8915.958} C_VEL
LIN {X 0,Y 440.566,Z 320.812,A -85,B 0,C 180,E1 -8917.101,E2 -8917.101} C_VEL
LIN {X 0,Y 441.272,Z 310.024,A -85,B 0,C 180,E1 -8918.24,E2 -8918.24} C_VEL
LIN {X 0,Y 441.772,Z 299.144,A -85,B 0,C 180,E1 -8919.153,E2 -8919.153} C_VEL
LIN {X 0,Y 442.313,Z 286.612,A -85,B 0,C 180,E1 -8919.97,E2 -8919.97} C_VEL
LIN {X 0,Y 442.686,Z 274.098,A -85,B 0,C 180,E1 -8920.576,E2 -8920.576} C_VEL
LIN {X 0,Y 443.009,Z 260.991,A -85,B 0,C 180,E1 -8921.002,E2 -8921.002} C_VEL
LIN {X 0,Y 443.265,Z 240.673,A -85,B 0,C 180,E1 -8921.372,E2 -8921.372} C_VEL
LIN {X 0,Y 443.839,Z 167.866,A -85,B 0,C 180,E1 -8922.552,E2 -8922.552} C_VEL
LIN {X 0,Y 440.558,Z 151.43,A -85,B 0,C 180,E1 -8922.961,E2 -8922.961} C_VEL
LIN {X 0,Y 440.607,Z 145.098,A -85,B 0,C 180,E1 -8924.313,E2 -8924.313} C_VEL
LIN {X 0,Y 439.507,Z 138.74,A -85,B 0,C 180,E1 -8925.773,E2 -8925.773} C_VEL
LIN {X 0,Y 439.441,Z 138.743,A -85,B 0,C 180,E1 -8929.336,E2 -8929.336} C_VEL
LIN {X 0,Y 439.364,Z 138.756,A -85,B 0,C 180,E1 -8932.574,E2 -8932.574} C_VEL
LIN {X 0,Y 439.396,Z 138.75,A -85,B 0,C 180,E1 -8935.584,E2 -8935.584} C_VEL
LIN {X 0,Y 439.415,Z 138.748,A -85,B 0,C 180,E1 -8938.672,E2 -8938.672} C_VEL
LIN {X 0,Y 439.368,Z 138.759,A -85,B 0,C 180,E1 -8942.029,E2 -8942.029} C_VEL
LIN {X 0,Y 439.391,Z 138.751,A -85,B 0,C 180,E1 -8945.339,E2 -8945.339} C_VEL
LIN {X 0,Y 439.381,Z 138.752,A -85,B 0,C 180,E1 -8948.593,E2 -8948.593} C_VEL
LIN {X 0,Y 439.384,Z 138.752,A -85,B 0,C 180,E1 -8951.255,E2 -8951.255} C_VEL
LIN {X 0,Y 439.394,Z 138.751,A -85,B 0,C 180,E1 -8954.728,E2 -8954.728} C_VEL
LIN {X 0,Y 439.389,Z 138.754,A -85,B 0,C 180,E1 -8957.794,E2 -8957.794} C_VEL
LIN {X 0,Y 439.387,Z 138.752,A -85,B 0,C 180,E1 -8960.223,E2 -8960.223} C_VEL
LIN {X 0,Y 439.365,Z 138.757,A -85,B 0,C 180,E1 -8963.712,E2 -8963.712} C_VEL
LIN {X 0,Y 439.363,Z 138.756,A -85,B 0,C 180,E1 -8967.053,E2 -8967.053} C_VEL
LIN {X 0,Y 439.372,Z 138.755,A -85,B 0,C 180,E1 -8970.273,E2 -8970.273} C_VEL
LIN {X 0,Y 439.409,Z 138.752,A -85,B 0,C 180,E1 -8973.395,E2 -8973.395} C_VEL
LIN {X 0,Y 439.37,Z 138.754,A -85,B 0,C 180,E1 -8976.428,E2 -8976.428} C_VEL
LIN {X 0,Y 439.376,Z 138.755,A -85,B 0,C 180,E1 -8979.396,E2 -8979.396} C_VEL
LIN {X 0,Y 439.388,Z 138.752,A -85,B 0,C 180,E1 -8982.308,E2 -8982.308} C_VEL
LIN {X 0,Y 439.422,Z 138.749,A -85,B 0,C 180,E1 -8985.173,E2 -8985.173} C_VEL
LIN {X 0,Y 439.471,Z 138.742,A -85,B 0,C 180,E1 -8988.001,E2 -8988.001} C_VEL
LIN {X 0,Y 439.491,Z 138.741,A -85,B 0,C 180,E1 -8991.725,E2 -8991.725} C_VEL
LIN {X 0,Y 439.584,Z 138.729,A -85,B 0,C 180,E1 -8994.495,E2 -8994.495} C_VEL
LIN {X 0,Y 439.613,Z 138.724,A -85,B 0,C 180,E1 -8998.168,E2 -8998.168} C_VEL
LIN {X 0,Y 439.655,Z 138.719,A -85,B 0,C 180,E1 -9000,E2 -9000} C_VEL
LIN {X 0,Y 439.592,Z 138.728,A -85,B 0,C 180,E1 -9002.749,E2 -9002.749} C_VEL
LIN {X 0,Y 439.55,Z 138.734,A -85,B 0,C 180,E1 -9006.426,E2 -9006.426} C_VEL
LIN {X 0,Y 439.481,Z 138.743,A -85,B 0,C 180,E1 -9009.202,E2 -9009.202} C_VEL
LIN {X 0,Y 439.453,Z 138.746,A -85,B 0,C 180,E1 -9012.938,E2 -9012.938} C_VEL
LIN {X 0,Y 439.434,Z 138.747,A -85,B 0,C 180,E1 -9016.348,E2 -9016.348} C_VEL
LIN {X 0,Y 439.39,Z 138.752,A -85,B 0,C 180,E1 -9019.627,E2 -9019.627} C_VEL
LIN {X 0,Y 439.35,Z 138.758,A -85,B 0,C 180,E1 -9022.576,E2 -9022.576} C_VEL
LIN {X 0,Y 439.375,Z 138.753,A -85,B 0,C 180,E1 -9025.587,E2 -9025.587} C_VEL
LIN {X 0,Y 439.407,Z 138.753,A -85,B 0,C 180,E1 -9028.674,E2 -9028.674} C_VEL
LIN {X 0,Y 439.358,Z 138.756,A -85,B 0,C 180,E1 -9032.031,E2 -9032.031} C_VEL
LIN {X 0,Y 439.383,Z 138.752,A -85,B 0,C 180,E1 -9035.341,E2 -9035.341} C_VEL
LIN {X 0,Y 439.367,Z 138.758,A -85,B 0,C 180,E1 -9038.597,E2 -9038.597} C_VEL
LIN {X 0,Y 439.38,Z 138.752,A -85,B 0,C 180,E1 -9041.258,E2 -9041.258} C_VEL
LIN {X 0,Y 439.392,Z 138.752,A -85,B 0,C 180,E1 -9044.731,E2 -9044.731} C_VEL
LIN {X 0,Y 439.389,Z 138.752,A -85,B 0,C 180,E1 -9047.797,E2 -9047.797} C_VEL
LIN {X 0,Y 439.431,Z 138.751,A -85,B 0,C 180,E1 -9050.23,E2 -9050.23} C_VEL
LIN {X 0,Y 439.369,Z 138.754,A -85,B 0,C 180,E1 -9053.714,E2 -9053.714} C_VEL
LIN {X 0,Y 439.368,Z 138.752,A -85,B 0,C 180,E1 -9057.055,E2 -9057.055} C_VEL
LIN {X 0,Y 439.379,Z 138.757,A -85,B 0,C 180,E1 -9060.275,E2 -9060.275} C_VEL
LIN {X 0,Y 439.492,Z 138.925,A -85,B 0,C 180,E1 -9062.953,E2 -9062.953} C_VEL
LIN {X 0,Y 441.777,Z 150.702,A -85,B 0,C 180,E1 -9065.244,E2 -9065.244} C_VEL
LIN {X 0,Y 441.862,Z 155.221,A -85,B 0,C 180,E1 -9066.073,E2 -9066.073} C_VEL
LIN {X 0,Y 440.92,Z 172.903,A -85,B 0,C 180,E1 -9069.229,E2 -9069.229} C_VEL
LIN {X 0,Y 440.214,Z 188.88,A -85,B 0,C 180,E1 -9072.054,E2 -9072.054} C_VEL
LIN {X 0,Y 443.607,Z 214.496,A -85,B 0,C 180,E1 -9072.603,E2 -9072.603} C_VEL
LIN {X 0,Y 442.887,Z 297.638,A -85,B 0,C 180,E1 -9073.967,E2 -9073.967} C_VEL
LIN {X 0,Y 442.36,Z 310.912,A -85,B 0,C 180,E1 -9074.361,E2 -9074.361} C_VEL
LIN {X 0,Y 441.905,Z 323.112,A -85,B 0,C 180,E1 -9074.906,E2 -9074.906} C_VEL
LIN {X 0,Y 441.302,Z 334.595,A -85,B 0,C 180,E1 -9075.592,E2 -9075.592} C_VEL
LIN {X 0,Y 440.625,Z 346.638,A -85,B 0,C 180,E1 -9076.534,E2 -9076.534} C_VEL
LIN {X 0,Y 440.06,Z 356.98,A -85,B 0,C 180,E1 -9077.55,E2 -9077.55} C_VEL
LIN {X 0,Y 439.585,Z 366.524,A -85,B 0,C 180,E1 -9078.707,E2 -9078.707} C_VEL
LIN {X 0,Y 439.022,Z 375.699,A -85,B 0,C 180,E1 -9080.092,E2 -9080.092} C_VEL
LIN {X 0,Y 438.701,Z 383.096,A -85,B 0,C 180,E1 -9081.479,E2 -9081.479} C_VEL
LIN {X 0,Y 438.496,Z 389.879,A -85,B 0,C 180,E1 -9083.097,E2 -9083.097} C_VEL
LIN {X 0,Y 438.374,Z 394.351,A -85,B 0,C 180,E1 -9084.481,E2 -9084.481} C_VEL
LIN {X 0,Y 438.342,Z 396.71,A -85,B 0,C 180,E1 -9085.403,E2 -9085.403} C_VEL
LIN {X 0,Y 438.319,Z 398.637,A -85,B 0,C 180,E1 -9086.324,E2 -9086.324} C_VEL
LIN {X 0,Y 438.381,Z 400.127,A -85,B 0,C 180,E1 -9087.244,E2 -9087.244} C_VEL
LIN {X 0,Y 438.31,Z 401.819,A -85,B 0,C 180,E1 -9089.082,E2 -9089.082} C_VEL
LIN {X 0,Y 438.317,Z 402.083,A -85,B 0,C 180,E1 -9090.001,E2 -9090.001} C_VEL
LIN {X 0,Y 438.311,Z 401.941,A -85,B 0,C 180,E1 -9090.92,E2 -9090.92} C_VEL
LIN {X 0,Y 438.375,Z 400.415,A -85,B 0,C 180,E1 -9092.758,E2 -9092.758} C_VEL
LIN {X 0,Y 438.292,Z 399.057,A -85,B 0,C 180,E1 -9093.678,E2 -9093.678} C_VEL
LIN {X 0,Y 438.375,Z 396.198,A -85,B 0,C 180,E1 -9095.059,E2 -9095.059} C_VEL
LIN {X 0,Y 438.369,Z 392.309,A -85,B 0,C 180,E1 -9096.444,E2 -9096.444} C_VEL
LIN {X 0,Y 438.599,Z 387.302,A -85,B 0,C 180,E1 -9097.829,E2 -9097.829} C_VEL
LIN {X 0,Y 438.898,Z 381.022,A -85,B 0,C 180,E1 -9099.215,E2 -9099.215} C_VEL
LIN {X 0,Y 439.324,Z 373.183,A -85,B 0,C 180,E1 -9100.602,E2 -9100.602} C_VEL
LIN {X 0,Y 439.938,Z 365.204,A -85,B 0,C 180,E1 -9101.753,E2 -9101.753} C_VEL
LIN {X 0,Y 440.485,Z 355.482,A -85,B 0,C 180,E1 -9102.908,E2 -9102.908} C_VEL
LIN {X 0,Y 441.157,Z 344.701,A -85,B 0,C 180,E1 -9103.944,E2 -9103.944} C_VEL
LIN {X 0,Y 441.828,Z 334.224,A -85,B 0,C 180,E1 -9104.745,E2 -9104.745} C_VEL
LIN {X 0,Y 442.504,Z 321.63,A -85,B 0,C 180,E1 -9105.488,E2 -9105.488} C_VEL
LIN {X 0,Y 443.136,Z 309.089,A -85,B 0,C 180,E1 -9106.026,E2 -9106.026} C_VEL
LIN {X 0,Y 443.615,Z 296.041,A -85,B 0,C 180,E1 -9106.392,E2 -9106.392} C_VEL
LIN {X 0,Y 444.348,Z 212.676,A -85,B 0,C 180,E1 -9107.768,E2 -9107.768} C_VEL
LIN {X 0,Y 440.561,Z 188.703,A -85,B 0,C 180,E1 -9108.345,E2 -9108.345} C_VEL
LIN {X 0,Y 441.62,Z 168.585,A -85,B 0,C 180,E1 -9111.962,E2 -9111.962} C_VEL
LIN {X 0,Y 442.422,Z 155.232,A -85,B 0,C 180,E1 -9114.395,E2 -9114.395} C_VEL
LIN {X 0,Y 441.799,Z 149.867,A -85,B 0,C 180,E1 -9115.437,E2 -9115.437} C_VEL
LIN {X 0,Y 439.457,Z 138.748,A -85,B 0,C 180,E1 -9117.749,E2 -9117.749} C_VEL
LIN {X 0,Y 439.363,Z 138.76,A -85,B 0,C 180,E1 -9120.789,E2 -9120.789} C_VEL
LIN {X 0,Y 439.39,Z 138.755,A -85,B 0,C 180,E1 -9124.044,E2 -9124.044} C_VEL
LIN {X 0,Y 439.349,Z 138.754,A -85,B 0,C 180,E1 -9126.887,E2 -9126.887} C_VEL
LIN {X 0,Y 439.404,Z 138.752,A -85,B 0,C 180,E1 -9129.849,E2 -9129.849} C_VEL
LIN {X 0,Y 439.372,Z 138.751,A -85,B 0,C 180,E1 -9132.625,E2 -9132.625} C_VEL
LIN {X 0,Y 439.4,Z 138.754,A -85,B 0,C 180,E1 -9135.27,E2 -9135.27} C_VEL
LIN {X 0,Y 439.371,Z 138.754,A -85,B 0,C 180,E1 -9138.746,E2 -9138.746} C_VEL
LIN {X 0,Y 439.366,Z 138.756,A -85,B 0,C 180,E1 -9141.609,E2 -9141.609} C_VEL
LIN {X 0,Y 439.397,Z 138.754,A -85,B 0,C 180,E1 -9144.844,E2 -9144.844} C_VEL
LIN {X 0,Y 439.371,Z 138.753,A -85,B 0,C 180,E1 -9148.139,E2 -9148.139} C_VEL
LIN {X 0,Y 439.401,Z 138.748,A -85,B 0,C 180,E1 -9151.606,E2 -9151.606} C_VEL
LIN {X 0,Y 439.366,Z 138.755,A -85,B 0,C 180,E1 -9154.413,E2 -9154.413} C_VEL
LIN {X 0,Y 439.36,Z 138.753,A -85,B 0,C 180,E1 -9157.424,E2 -9157.424} C_VEL
LIN {X 0,Y 439.441,Z 138.742,A -85,B 0,C 180,E1 -9160.664,E2 -9160.664} C_VEL
LIN {X 0,Y 439.418,Z 138.75,A -85,B 0,C 180,E1 -9164.223,E2 -9164.223} C_VEL
LIN {X 0,Y 439.484,Z 138.736,A -85,B 0,C 180,E1 -9167.286,E2 -9167.286} C_VEL
LIN {X 0,Y 439.471,Z 138.734,A -85,B 0,C 180,E1 -9170.798,E2 -9170.798} C_VEL
LIN {X 0,Y 439.556,Z 138.729,A -85,B 0,C 180,E1 -9173.574,E2 -9173.574} C_VEL
LIN {X 0,Y 439.399,Z 138.749,A -85,B 0,C 180,E1 -9175.413,E2 -9175.413} C_VEL
LIN {X 0,Y 439.624,Z 138.723,A -85,B 0,C 180,E1 -9178.168,E2 -9178.168} C_VEL
LIN {X 0,Y 439.667,Z 138.721,A -85,B 0,C 180,E1 -9180,E2 -9180} C_VEL
LIN {X 0,Y 439.603,Z 138.716,A -85,B 0,C 180,E1 -9182.749,E2 -9182.749} C_VEL
LIN {X 0,Y 439.558,Z 138.728,A -85,B 0,C 180,E1 -9186.426,E2 -9186.426} C_VEL
LIN {X 0,Y 439.493,Z 138.732,A -85,B 0,C 180,E1 -9189.202,E2 -9189.202} C_VEL
LIN {X 0,Y 439.466,Z 138.741,A -85,B 0,C 180,E1 -9192.938,E2 -9192.938} C_VEL
LIN {X 0,Y 439.447,Z 138.742,A -85,B 0,C 180,E1 -9196.348,E2 -9196.348} C_VEL
LIN {X 0,Y 439.403,Z 138.747,A -85,B 0,C 180,E1 -9199.626,E2 -9199.626} C_VEL
LIN {X 0,Y 439.363,Z 138.754,A -85,B 0,C 180,E1 -9202.576,E2 -9202.576} C_VEL
LIN {X 0,Y 439.378,Z 138.752,A -85,B 0,C 180,E1 -9205.587,E2 -9205.587} C_VEL
LIN {X 0,Y 439.401,Z 138.75,A -85,B 0,C 180,E1 -9208.675,E2 -9208.675} C_VEL
LIN {X 0,Y 439.37,Z 138.751,A -85,B 0,C 180,E1 -9212.03,E2 -9212.03} C_VEL
LIN {X 0,Y 439.394,Z 138.749,A -85,B 0,C 180,E1 -9215.34,E2 -9215.34} C_VEL
LIN {X 0,Y 439.372,Z 138.756,A -85,B 0,C 180,E1 -9218.596,E2 -9218.596} C_VEL
LIN {X 0,Y 439.391,Z 138.74,A -85,B 0,C 180,E1 -9221.257,E2 -9221.257} C_VEL
LIN {X 0,Y 439.402,Z 138.75,A -85,B 0,C 180,E1 -9224.73,E2 -9224.73} C_VEL
LIN {X 0,Y 439.387,Z 138.752,A -85,B 0,C 180,E1 -9227.794,E2 -9227.794} C_VEL
LIN {X 0,Y 439.392,Z 138.756,A -85,B 0,C 180,E1 -9230.223,E2 -9230.223} C_VEL
LIN {X 0,Y 439.378,Z 138.755,A -85,B 0,C 180,E1 -9233.713,E2 -9233.713} C_VEL
LIN {X 0,Y 439.376,Z 138.752,A -85,B 0,C 180,E1 -9237.054,E2 -9237.054} C_VEL
LIN {X 0,Y 439.386,Z 138.753,A -85,B 0,C 180,E1 -9240.274,E2 -9240.274} C_VEL
LIN {X 0,Y 439.433,Z 138.751,A -85,B 0,C 180,E1 -9243.396,E2 -9243.396} C_VEL
LIN {X 0,Y 439.459,Z 138.803,A -85,B 0,C 180,E1 -9243.808,E2 -9243.808} C_VEL
LIN {X 0,Y 441.007,Z 147.251,A -85,B 0,C 180,E1 -9245.772,E2 -9245.772} C_VEL
LIN {X 0,Y 441.056,Z 151.575,A -85,B 0,C 180,E1 -9246.715,E2 -9246.715} C_VEL
LIN {X 0,Y 444.826,Z 168.515,A -85,B 0,C 180,E1 -9247.191,E2 -9247.191} C_VEL
LIN {X 0,Y 443.852,Z 259.333,A -85,B 0,C 180,E1 -9248.698,E2 -9248.698} C_VEL
LIN {X 0,Y 443.452,Z 272.264,A -85,B 0,C 180,E1 -9249.094,E2 -9249.094} C_VEL
LIN {X 0,Y 443.032,Z 284.145,A -85,B 0,C 180,E1 -9249.634,E2 -9249.634} C_VEL
LIN {X 0,Y 442.493,Z 296.477,A -85,B 0,C 180,E1 -9250.395,E2 -9250.395} C_VEL
LIN {X 0,Y 441.733,Z 308.087,A -85,B 0,C 180,E1 -9251.325,E2 -9251.325} C_VEL
LIN {X 0,Y 441.457,Z 313.606,A -85,B 0,C 180,E1 -9251.856,E2 -9251.856} C_VEL
LIN {X 0,Y 440.506,Z 318.249,A -85,B 0,C 180,E1 -9252.317,E2 -9252.317} C_VEL
LIN {X 0,Y 437.271,Z 325.517,A -85,B 0,C 180,E1 -9253.092,E2 -9253.092} C_VEL
LIN {X 0,Y 434.021,Z 332.201,A -85,B 0,C 180,E1 -9253.955,E2 -9253.955} C_VEL
LIN {X 0,Y 433.058,Z 335.925,A -85,B 0,C 180,E1 -9254.548,E2 -9254.548} C_VEL
LIN {X 0,Y 432.495,Z 342.99,A -85,B 0,C 180,E1 -9255.891,E2 -9255.891} C_VEL
LIN {X 0,Y 432.045,Z 349.434,A -85,B 0,C 180,E1 -9257.426,E2 -9257.426} C_VEL
LIN {X 0,Y 431.77,Z 353.751,A -85,B 0,C 180,E1 -9258.736,E2 -9258.736} C_VEL
LIN {X 0,Y 431.493,Z 357.371,A -85,B 0,C 180,E1 -9260.152,E2 -9260.152} C_VEL
LIN {X 0,Y 431.381,Z 359.967,A -85,B 0,C 180,E1 -9261.568,E2 -9261.568} C_VEL
LIN {X 0,Y 431.374,Z 361.183,A -85,B 0,C 180,E1 -9262.51,E2 -9262.51} C_VEL
LIN {X 0,Y 431.381,Z 362.066,A -85,B 0,C 180,E1 -9263.621,E2 -9263.621} C_VEL
LIN {X 0,Y 431.269,Z 362.366,A -85,B 0,C 180,E1 -9265.326,E2 -9265.326} C_VEL
LIN {X 0,Y 431.302,Z 361.988,A -85,B 0,C 180,E1 -9266.262,E2 -9266.262} C_VEL
LIN {X 0,Y 431.354,Z 361.207,A -85,B 0,C 180,E1 -9267.198,E2 -9267.198} C_VEL
LIN {X 0,Y 431.333,Z 358.409,A -85,B 0,C 180,E1 -9269.066,E2 -9269.066} C_VEL
LIN {X 0,Y 431.48,Z 355.201,A -85,B 0,C 180,E1 -9270.466,E2 -9270.466} C_VEL
LIN {X 0,Y 431.607,Z 350.949,A -85,B 0,C 180,E1 -9271.865,E2 -9271.865} C_VEL
LIN {X 0,Y 431.976,Z 345.516,A -85,B 0,C 180,E1 -9273.263,E2 -9273.263} C_VEL
LIN {X 0,Y 432.4,Z 338.742,A -85,B 0,C 180,E1 -9274.66,E2 -9274.66} C_VEL
LIN {X 0,Y 433.054,Z 330.273,A -85,B 0,C 180,E1 -9276.054,E2 -9276.054} C_VEL
LIN {X 0,Y 433.572,Z 321.596,A -85,B 0,C 180,E1 -9277.216,E2 -9277.216} C_VEL
LIN {X 0,Y 434.313,Z 310.903,A -85,B 0,C 180,E1 -9278.373,E2 -9278.373} C_VEL
LIN {X 0,Y 434.825,Z 300.211,A -85,B 0,C 180,E1 -9279.3,E2 -9279.3} C_VEL
LIN {X 0,Y 435.408,Z 287.637,A -85,B 0,C 180,E1 -9280.144,E2 -9280.144} C_VEL
LIN {X 0,Y 435.775,Z 275.707,A -85,B 0,C 180,E1 -9280.746,E2 -9280.746} C_VEL
LIN {X 0,Y 436.125,Z 263.447,A -85,B 0,C 180,E1 -9281.178,E2 -9281.178} C_VEL
LIN {X 0,Y 436.303,Z 247.91,A -85,B 0,C 180,E1 -9281.497,E2 -9281.497} C_VEL
LIN {X 0,Y 437.097,Z 170.105,A -85,B 0,C 180,E1 -9282.772,E2 -9282.772} C_VEL
LIN {X 0,Y 433.612,Z 151.696,A -85,B 0,C 180,E1 -9283.237,E2 -9283.237} C_VEL
LIN {X 0,Y 433.575,Z 145.651,A -85,B 0,C 180,E1 -9284.55,E2 -9284.55} C_VEL
LIN {X 0,Y 432.453,Z 139.619,A -85,B 0,C 180,E1 -9285.976,E2 -9285.976} C_VEL
LIN {X 0,Y 432.387,Z 139.623,A -85,B 0,C 180,E1 -9289.484,E2 -9289.484} C_VEL
LIN {X 0,Y 432.318,Z 139.631,A -85,B 0,C 180,E1 -9292.963,E2 -9292.963} C_VEL
LIN {X 0,Y 432.36,Z 139.63,A -85,B 0,C 180,E1 -9296.031,E2 -9296.031} C_VEL
LIN {X 0,Y 432.341,Z 139.628,A -85,B 0,C 180,E1 -9299.186,E2 -9299.186} C_VEL
LIN {X 0,Y 432.32,Z 139.633,A -85,B 0,C 180,E1 -9302.442,E2 -9302.442} C_VEL
LIN {X 0,Y 432.341,Z 139.631,A -85,B 0,C 180,E1 -9305.631,E2 -9305.631} C_VEL
LIN {X 0,Y 432.35,Z 139.628,A -85,B 0,C 180,E1 -9309.341,E2 -9309.341} C_VEL
LIN {X 0,Y 432.329,Z 139.635,A -85,B 0,C 180,E1 -9311.796,E2 -9311.796} C_VEL
LIN {X 0,Y 432.328,Z 139.631,A -85,B 0,C 180,E1 -9314.346,E2 -9314.346} C_VEL
LIN {X 0,Y 432.313,Z 139.633,A -85,B 0,C 180,E1 -9317.015,E2 -9317.015} C_VEL
LIN {X 0,Y 432.326,Z 139.634,A -85,B 0,C 180,E1 -9319.82,E2 -9319.82} C_VEL
LIN {X 0,Y 432.298,Z 139.635,A -85,B 0,C 180,E1 -9323.021,E2 -9323.021} C_VEL
LIN {X 0,Y 432.349,Z 139.629,A -85,B 0,C 180,E1 -9325.996,E2 -9325.996} C_VEL
LIN {X 0,Y 432.338,Z 139.633,A -85,B 0,C 180,E1 -9329.489,E2 -9329.489} C_VEL
LIN {X 0,Y 432.375,Z 139.626,A -85,B 0,C 180,E1 -9332.927,E2 -9332.927} C_VEL
LIN {X 0,Y 432.354,Z 139.63,A -85,B 0,C 180,E1 -9336.022,E2 -9336.022} C_VEL
LIN {X 0,Y 432.339,Z 139.633,A -85,B 0,C 180,E1 -9339.045,E2 -9339.045} C_VEL
LIN {X 0,Y 432.345,Z 139.63,A -85,B 0,C 180,E1 -9342.01,E2 -9342.01} C_VEL
LIN {X 0,Y 432.369,Z 139.629,A -85,B 0,C 180,E1 -9344.925,E2 -9344.925} C_VEL
LIN {X 0,Y 432.447,Z 139.618,A -85,B 0,C 180,E1 -9347.803,E2 -9347.803} C_VEL
LIN {X 0,Y 432.451,Z 139.618,A -85,B 0,C 180,E1 -9351.589,E2 -9351.589} C_VEL
LIN {X 0,Y 432.539,Z 139.606,A -85,B 0,C 180,E1 -9354.405,E2 -9354.405} C_VEL
LIN {X 0,Y 432.582,Z 139.6,A -85,B 0,C 180,E1 -9358.138,E2 -9358.138} C_VEL
LIN {X 0,Y 432.607,Z 139.597,A -85,B 0,C 180,E1 -9360,E2 -9360} C_VEL
LIN {X 0,Y 432.546,Z 139.606,A -85,B 0,C 180,E1 -9362.794,E2 -9362.794} C_VEL
LIN {X 0,Y 432.561,Z 139.603,A -85,B 0,C 180,E1 -9365.594,E2 -9365.594} C_VEL
LIN {X 0,Y 432.451,Z 139.618,A -85,B 0,C 180,E1 -9368.41,E2 -9368.41} C_VEL
LIN {X 0,Y 432.447,Z 139.618,A -85,B 0,C 180,E1 -9372.197,E2 -9372.197} C_VEL
LIN {X 0,Y 432.417,Z 139.621,A -85,B 0,C 180,E1 -9376.039,E2 -9376.039} C_VEL
LIN {X 0,Y 432.375,Z 139.625,A -85,B 0,C 180,E1 -9379.485,E2 -9379.485} C_VEL
LIN {X 0,Y 432.304,Z 139.637,A -85,B 0,C 180,E1 -9382.965,E2 -9382.965} C_VEL
LIN {X 0,Y 432.339,Z 139.631,A -85,B 0,C 180,E1 -9386.034,E2 -9386.034} C_VEL
LIN {X 0,Y 432.332,Z 139.631,A -85,B 0,C 180,E1 -9389.188,E2 -9389.188} C_VEL
LIN {X 0,Y 432.313,Z 139.636,A -85,B 0,C 180,E1 -9392.444,E2 -9392.444} C_VEL
LIN {X 0,Y 432.334,Z 139.63,A -85,B 0,C 180,E1 -9395.632,E2 -9395.632} C_VEL
LIN {X 0,Y 432.329,Z 139.633,A -85,B 0,C 180,E1 -9398.715,E2 -9398.715} C_VEL
LIN {X 0,Y 432.325,Z 139.631,A -85,B 0,C 180,E1 -9401.798,E2 -9401.798} C_VEL
LIN {X 0,Y 432.326,Z 139.636,A -85,B 0,C 180,E1 -9404.348,E2 -9404.348} C_VEL
LIN {X 0,Y 432.313,Z 139.632,A -85,B 0,C 180,E1 -9407.017,E2 -9407.017} C_VEL
LIN {X 0,Y 432.335,Z 139.631,A -85,B 0,C 180,E1 -9409.821,E2 -9409.821} C_VEL
LIN {X 0,Y 432.301,Z 139.633,A -85,B 0,C 180,E1 -9413.023,E2 -9413.023} C_VEL
LIN {X 0,Y 432.355,Z 139.632,A -85,B 0,C 180,E1 -9415.998,E2 -9415.998} C_VEL
LIN {X 0,Y 432.344,Z 139.629,A -85,B 0,C 180,E1 -9419.491,E2 -9419.491} C_VEL
LIN {X 0,Y 432.449,Z 139.787,A -85,B 0,C 180,E1 -9422.737,E2 -9422.737} C_VEL
LIN {X 0,Y 434.823,Z 151.978,A -85,B 0,C 180,E1 -9425.152,E2 -9425.152} C_VEL
LIN {X 0,Y 434.855,Z 157.459,A -85,B 0,C 180,E1 -9426.17,E2 -9426.17} C_VEL
LIN {X 0,Y 433.826,Z 175.13,A -85,B 0,C 180,E1 -9429.37,E2 -9429.37} C_VEL
LIN {X 0,Y 433.262,Z 188.502,A -85,B 0,C 180,E1 -9431.775,E2 -9431.775} C_VEL
LIN {X 0,Y 436.766,Z 214.373,A -85,B 0,C 180,E1 -9432.352,E2 -9432.352} C_VEL
LIN {X 0,Y 436.007,Z 297.448,A -85,B 0,C 180,E1 -9433.737,E2 -9433.737} C_VEL
LIN {X 0,Y 435.49,Z 310.683,A -85,B 0,C 180,E1 -9434.138,E2 -9434.138} C_VEL
LIN {X 0,Y 434.976,Z 323.427,A -85,B 0,C 180,E1 -9434.719,E2 -9434.719} C_VEL
LIN {X 0,Y 434.295,Z 335.529,A -85,B 0,C 180,E1 -9435.474,E2 -9435.474} C_VEL
LIN {X 0,Y 433.623,Z 347.046,A -85,B 0,C 180,E1 -9436.405,E2 -9436.405} C_VEL
LIN {X 0,Y 433.018,Z 357.5,A -85,B 0,C 180,E1 -9437.463,E2 -9437.463} C_VEL
LIN {X 0,Y 432.554,Z 366.013,A -85,B 0,C 180,E1 -9438.521,E2 -9438.521} C_VEL
LIN {X 0,Y 431.976,Z 375.228,A -85,B 0,C 180,E1 -9439.928,E2 -9439.928} C_VEL
LIN {X 0,Y 431.645,Z 382.653,A -85,B 0,C 180,E1 -9441.339,E2 -9441.339} C_VEL
LIN {X 0,Y 431.412,Z 389.469,A -85,B 0,C 180,E1 -9442.983,E2 -9442.983} C_VEL
LIN {X 0,Y 431.274,Z 393.961,A -85,B 0,C 180,E1 -9444.39,E2 -9444.39} C_VEL
LIN {X 0,Y 431.274,Z 396.332,A -85,B 0,C 180,E1 -9445.327,E2 -9445.327} C_VEL
LIN {X 0,Y 431.222,Z 398.267,A -85,B 0,C 180,E1 -9446.263,E2 -9446.263} C_VEL
LIN {X 0,Y 431.308,Z 399.774,A -85,B 0,C 180,E1 -9447.199,E2 -9447.199} C_VEL
LIN {X 0,Y 431.224,Z 401.483,A -85,B 0,C 180,E1 -9449.067,E2 -9449.067} C_VEL
LIN {X 0,Y 431.228,Z 401.755,A -85,B 0,C 180,E1 -9450.001,E2 -9450.001} C_VEL
LIN {X 0,Y 431.224,Z 401.628,A -85,B 0,C 180,E1 -9450.935,E2 -9450.935} C_VEL
LIN {X 0,Y 431.283,Z 400.12,A -85,B 0,C 180,E1 -9452.803,E2 -9452.803} C_VEL
LIN {X 0,Y 431.197,Z 398.769,A -85,B 0,C 180,E1 -9453.739,E2 -9453.739} C_VEL
LIN {X 0,Y 431.283,Z 395.928,A -85,B 0,C 180,E1 -9455.143,E2 -9455.143} C_VEL
LIN {X 0,Y 431.291,Z 392.058,A -85,B 0,C 180,E1 -9456.551,E2 -9456.551} C_VEL
LIN {X 0,Y 431.532,Z 387.072,A -85,B 0,C 180,E1 -9457.958,E2 -9457.958} C_VEL
LIN {X 0,Y 431.837,Z 380.815,A -85,B 0,C 180,E1 -9459.367,E2 -9459.367} C_VEL
LIN {X 0,Y 432.316,Z 373.018,A -85,B 0,C 180,E1 -9460.776,E2 -9460.776} C_VEL
LIN {X 0,Y 432.949,Z 365.071,A -85,B 0,C 180,E1 -9461.945,E2 -9461.945} C_VEL
LIN {X 0,Y 433.538,Z 355.39,A -85,B 0,C 180,E1 -9463.118,E2 -9463.118} C_VEL
LIN {X 0,Y 434.26,Z 344.66,A -85,B 0,C 180,E1 -9464.17,E2 -9464.17} C_VEL
LIN {X 0,Y 434.963,Z 334.27,A -85,B 0,C 180,E1 -9464.983,E2 -9464.983} C_VEL
LIN {X 0,Y 435.688,Z 321.808,A -85,B 0,C 180,E1 -9465.736,E2 -9465.736} C_VEL
LIN {X 0,Y 436.344,Z 309.444,A -85,B 0,C 180,E1 -9466.282,E2 -9466.282} C_VEL
LIN {X 0,Y 436.847,Z 296.926,A -85,B 0,C 180,E1 -9466.653,E2 -9466.653} C_VEL
LIN {X 0,Y 437.648,Z 213.585,A -85,B 0,C 180,E1 -9468.056,E2 -9468.056} C_VEL
LIN {X 0,Y 433.984,Z 190.38,A -85,B 0,C 180,E1 -9468.626,E2 -9468.626} C_VEL
LIN {X 0,Y 433.638,Z 188.227,A -85,B 0,C 180,E1 -9468.703,E2 -9468.703} C_VEL
LIN {X 0,Y 434.76,Z 168.419,A -85,B 0,C 180,E1 -9472.327,E2 -9472.327} C_VEL
LIN {X 0,Y 435.517,Z 156.408,A -85,B 0,C 180,E1 -9474.553,E2 -9474.553} C_VEL
LIN {X 0,Y 434.962,Z 151.679,A -85,B 0,C 180,E1 -9475.488,E2 -9475.488} C_VEL
LIN {X 0,Y 432.402,Z 139.627,A -85,B 0,C 180,E1 -9477.99,E2 -9477.99} C_VEL
LIN {X 0,Y 432.324,Z 139.638,A -85,B 0,C 180,E1 -9481.346,E2 -9481.346} C_VEL
LIN {X 0,Y 432.342,Z 139.627,A -85,B 0,C 180,E1 -9484.677,E2 -9484.677} C_VEL
LIN {X 0,Y 432.334,Z 139.629,A -85,B 0,C 180,E1 -9488.151,E2 -9488.151} C_VEL
LIN {X 0,Y 432.326,Z 139.634,A -85,B 0,C 180,E1 -9491.601,E2 -9491.601} C_VEL
LIN {X 0,Y 432.335,Z 139.629,A -85,B 0,C 180,E1 -9494.347,E2 -9494.347} C_VEL
LIN {X 0,Y 432.318,Z 139.634,A -85,B 0,C 180,E1 -9497.016,E2 -9497.016} C_VEL
LIN {X 0,Y 432.292,Z 139.636,A -85,B 0,C 180,E1 -9499.828,E2 -9499.828} C_VEL
LIN {X 0,Y 432.307,Z 139.637,A -85,B 0,C 180,E1 -9503.022,E2 -9503.022} C_VEL
LIN {X 0,Y 432.334,Z 139.629,A -85,B 0,C 180,E1 -9506.002,E2 -9506.002} C_VEL
LIN {X 0,Y 432.347,Z 139.629,A -85,B 0,C 180,E1 -9509.49,E2 -9509.49} C_VEL
LIN {X 0,Y 432.335,Z 139.627,A -85,B 0,C 180,E1 -9511.873,E2 -9511.873} C_VEL
LIN {X 0,Y 432.324,Z 139.634,A -85,B 0,C 180,E1 -9514.997,E2 -9514.997} C_VEL
LIN {X 0,Y 432.355,Z 139.627,A -85,B 0,C 180,E1 -9518.046,E2 -9518.046} C_VEL
LIN {X 0,Y 432.381,Z 139.622,A -85,B 0,C 180,E1 -9521.029,E2 -9521.029} C_VEL
LIN {X 0,Y 432.388,Z 139.623,A -85,B 0,C 180,E1 -9523.96,E2 -9523.96} C_VEL
LIN {X 0,Y 432.452,Z 139.614,A -85,B 0,C 180,E1 -9527.803,E2 -9527.803} C_VEL
LIN {X 0,Y 432.445,Z 139.609,A -85,B 0,C 180,E1 -9531.589,E2 -9531.589} C_VEL
LIN {X 0,Y 432.548,Z 139.605,A -85,B 0,C 180,E1 -9534.406,E2 -9534.406} C_VEL
LIN {X 0,Y 432.594,Z 139.597,A -85,B 0,C 180,E1 -9538.138,E2 -9538.138} C_VEL
LIN {X 0,Y 432.619,Z 139.599,A -85,B 0,C 180,E1 -9540,E2 -9540} C_VEL
LIN {X 0,Y 432.556,Z 139.593,A -85,B 0,C 180,E1 -9542.794,E2 -9542.794} C_VEL
LIN {X 0,Y 432.569,Z 139.604,A -85,B 0,C 180,E1 -9545.594,E2 -9545.594} C_VEL
LIN {X 0,Y 432.463,Z 139.605,A -85,B 0,C 180,E1 -9548.41,E2 -9548.41} C_VEL
LIN {X 0,Y 432.459,Z 139.613,A -85,B 0,C 180,E1 -9552.197,E2 -9552.197} C_VEL
LIN {X 0,Y 432.43,Z 139.617,A -85,B 0,C 180,E1 -9556.039,E2 -9556.039} C_VEL
LIN {X 0,Y 432.388,Z 139.621,A -85,B 0,C 180,E1 -9559.485,E2 -9559.485} C_VEL
LIN {X 0,Y 432.317,Z 139.636,A -85,B 0,C 180,E1 -9562.965,E2 -9562.965} C_VEL
LIN {X 0,Y 432.338,Z 139.628,A -85,B 0,C 180,E1 -9565.002,E2 -9565.002} C_VEL
LIN {X 0,Y 432.348,Z 139.625,A -85,B 0,C 180,E1 -9568.126,E2 -9568.126} C_VEL
LIN {X 0,Y 432.322,Z 139.631,A -85,B 0,C 180,E1 -9571.346,E2 -9571.346} C_VEL
LIN {X 0,Y 432.339,Z 139.634,A -85,B 0,C 180,E1 -9574.677,E2 -9574.677} C_VEL
LIN {X 0,Y 432.335,Z 139.63,A -85,B 0,C 180,E1 -9578.15,E2 -9578.15} C_VEL
LIN {X 0,Y 432.335,Z 139.618,A -85,B 0,C 180,E1 -9581.602,E2 -9581.602} C_VEL
LIN {X 0,Y 432.337,Z 139.634,A -85,B 0,C 180,E1 -9584.347,E2 -9584.347} C_VEL
LIN {X 0,Y 432.319,Z 139.631,A -85,B 0,C 180,E1 -9587.016,E2 -9587.016} C_VEL
LIN {X 0,Y 432.335,Z 139.632,A -85,B 0,C 180,E1 -9589.821,E2 -9589.821} C_VEL
LIN {X 0,Y 432.31,Z 139.632,A -85,B 0,C 180,E1 -9593.022,E2 -9593.022} C_VEL
LIN {X 0,Y 432.363,Z 139.63,A -85,B 0,C 180,E1 -9595.996,E2 -9595.996} C_VEL
LIN {X 0,Y 432.352,Z 139.631,A -85,B 0,C 180,E1 -9599.489,E2 -9599.489} C_VEL
LIN {X 0,Y 432.396,Z 139.626,A -85,B 0,C 180,E1 -9602.928,E2 -9602.928} C_VEL
LIN {X 0,Y 432.418,Z 139.735,A -85,B 0,C 180,E1 -9603.566,E2 -9603.566} C_VEL
LIN {X 0,Y 434.049,Z 148.418,A -85,B 0,C 180,E1 -9605.613,E2 -9605.613} C_VEL
LIN {X 0,Y 434.187,Z 151.978,A -85,B 0,C 180,E1 -9606.398,E2 -9606.398} C_VEL
LIN {X 0,Y 438.101,Z 169.142,A -85,B 0,C 180,E1 -9606.885,E2 -9606.885} C_VEL
LIN {X 0,Y 437.148,Z 258.827,A -85,B 0,C 180,E1 -9608.391,E2 -9608.391} C_VEL
LIN {X 0,Y 436.723,Z 272.255,A -85,B 0,C 180,E1 -9608.802,E2 -9608.802} C_VEL
LIN {X 0,Y 436.253,Z 284.532,A -85,B 0,C 180,E1 -9609.365,E2 -9609.365} C_VEL
LIN {X 0,Y 435.749,Z 296.041,A -85,B 0,C 180,E1 -9610.079,E2 -9610.079} C_VEL
LIN {X 0,Y 434.945,Z 307.796,A -85,B 0,C 180,E1 -9611.022,E2 -9611.022} C_VEL
LIN {X 0,Y 434.314,Z 318.326,A -85,B 0,C 180,E1 -9612.093,E2 -9612.093} C_VEL
LIN {X 0,Y 433.687,Z 327.766,A -85,B 0,C 180,E1 -9613.282,E2 -9613.282} C_VEL
LIN {X 0,Y 433.058,Z 335.925,A -85,B 0,C 180,E1 -9614.548,E2 -9614.548} C_VEL
LIN {X 0,Y 432.097,Z 339.501,A -85,B 0,C 180,E1 -9615.166,E2 -9615.166} C_VEL
LIN {X 0,Y 428.855,Z 344.931,A -85,B 0,C 180,E1 -9616.187,E2 -9616.187} C_VEL
LIN {X 0,Y 425.69,Z 349.669,A -85,B 0,C 180,E1 -9617.271,E2 -9617.271} C_VEL
LIN {X 0,Y 424.853,Z 352.177,A -85,B 0,C 180,E1 -9617.978,E2 -9617.978} C_VEL
LIN {X 0,Y 424.513,Z 356.491,A -85,B 0,C 180,E1 -9619.507,E2 -9619.507} C_VEL
LIN {X 0,Y 424.392,Z 358.567,A -85,B 0,C 180,E1 -9620.467,E2 -9620.467} C_VEL
LIN {X 0,Y 424.291,Z 361.441,A -85,B 0,C 180,E1 -9622.384,E2 -9622.384} C_VEL
LIN {X 0,Y 424.305,Z 362.417,A -85,B 0,C 180,E1 -9623.627,E2 -9623.627} C_VEL
LIN {X 0,Y 424.197,Z 362.699,A -85,B 0,C 180,E1 -9625.247,E2 -9625.247} C_VEL
LIN {X 0,Y 424.282,Z 361.591,A -85,B 0,C 180,E1 -9627.151,E2 -9627.151} C_VEL
LIN {X 0,Y 424.243,Z 358.838,A -85,B 0,C 180,E1 -9629.05,E2 -9629.05} C_VEL
LIN {X 0,Y 424.403,Z 355.67,A -85,B 0,C 180,E1 -9630.474,E2 -9630.474} C_VEL
LIN {X 0,Y 424.547,Z 351.46,A -85,B 0,C 180,E1 -9631.896,E2 -9631.896} C_VEL
LIN {X 0,Y 425.047,Z 345.073,A -85,B 0,C 180,E1 -9633.554,E2 -9633.554} C_VEL
LIN {X 0,Y 425.459,Z 338.09,A -85,B 0,C 180,E1 -9634.974,E2 -9634.974} C_VEL
LIN {X 0,Y 426.136,Z 329.366,A -85,B 0,C 180,E1 -9636.391,E2 -9636.391} C_VEL
LIN {X 0,Y 426.735,Z 320.44,A -85,B 0,C 180,E1 -9637.57,E2 -9637.57} C_VEL
LIN {X 0,Y 427.421,Z 310.603,A -85,B 0,C 180,E1 -9638.628,E2 -9638.628} C_VEL
LIN {X 0,Y 427.973,Z 299.665,A -85,B 0,C 180,E1 -9639.573,E2 -9639.573} C_VEL
LIN {X 0,Y 428.553,Z 287.494,A -85,B 0,C 180,E1 -9640.392,E2 -9640.392} C_VEL
LIN {X 0,Y 428.905,Z 275.948,A -85,B 0,C 180,E1 -9640.98,E2 -9640.98} C_VEL
LIN {X 0,Y 429.275,Z 263.625,A -85,B 0,C 180,E1 -9641.419,E2 -9641.419} C_VEL
LIN {X 0,Y 429.464,Z 248,A -85,B 0,C 180,E1 -9641.743,E2 -9641.743} C_VEL
LIN {X 0,Y 430.307,Z 171.932,A -85,B 0,C 180,E1 -9643.007,E2 -9643.007} C_VEL
LIN {X 0,Y 429.578,Z 166.572,A -85,B 0,C 180,E1 -9643.127,E2 -9643.127} C_VEL
LIN {X 0,Y 426.673,Z 152.066,A -85,B 0,C 180,E1 -9643.497,E2 -9643.497} C_VEL
LIN {X 0,Y 426.65,Z 147.285,A -85,B 0,C 180,E1 -9644.548,E2 -9644.548} C_VEL
LIN {X 0,Y 425.397,Z 140.499,A -85,B 0,C 180,E1 -9646.125,E2 -9646.125} C_VEL
LIN {X 0,Y 425.329,Z 140.503,A -85,B 0,C 180,E1 -9649.634,E2 -9649.634} C_VEL
LIN {X 0,Y 425.288,Z 140.512,A -85,B 0,C 180,E1 -9652.337,E2 -9652.337} C_VEL
LIN {X 0,Y 425.29,Z 140.506,A -85,B 0,C 180,E1 -9655.444,E2 -9655.444} C_VEL
LIN {X 0,Y 425.347,Z 140.5,A -85,B 0,C 180,E1 -9657.556,E2 -9657.556} C_VEL
LIN {X 0,Y 425.286,Z 140.508,A -85,B 0,C 180,E1 -9660.815,E2 -9660.815} C_VEL
LIN {X 0,Y 425.308,Z 140.507,A -85,B 0,C 180,E1 -9664.287,E2 -9664.287} C_VEL
LIN {X 0,Y 425.276,Z 140.512,A -85,B 0,C 180,E1 -9667.693,E2 -9667.693} C_VEL
LIN {X 0,Y 425.279,Z 140.509,A -85,B 0,C 180,E1 -9670.52,E2 -9670.52} C_VEL
LIN {X 0,Y 425.252,Z 140.513,A -85,B 0,C 180,E1 -9673.35,E2 -9673.35} C_VEL
LIN {X 0,Y 425.25,Z 140.512,A -85,B 0,C 180,E1 -9676.648,E2 -9676.648} C_VEL
LIN {X 0,Y 425.278,Z 140.511,A -85,B 0,C 180,E1 -9679.871,E2 -9679.871} C_VEL
LIN {X 0,Y 425.269,Z 140.51,A -85,B 0,C 180,E1 -9682.488,E2 -9682.488} C_VEL
LIN {X 0,Y 425.297,Z 140.509,A -85,B 0,C 180,E1 -9685.816,E2 -9685.816} C_VEL
LIN {X 0,Y 425.281,Z 140.511,A -85,B 0,C 180,E1 -9689.238,E2 -9689.238} C_VEL
LIN {X 0,Y 425.336,Z 140.502,A -85,B 0,C 180,E1 -9692.441,E2 -9692.441} C_VEL
LIN {X 0,Y 425.335,Z 140.504,A -85,B 0,C 180,E1 -9695.601,E2 -9695.601} C_VEL
LIN {X 0,Y 425.281,Z 140.509,A -85,B 0,C 180,E1 -9698.681,E2 -9698.681} C_VEL
LIN {X 0,Y 425.307,Z 140.507,A -85,B 0,C 180,E1 -9701.701,E2 -9701.701} C_VEL
LIN {X 0,Y 425.323,Z 140.505,A -85,B 0,C 180,E1 -9704.67,E2 -9704.67} C_VEL
LIN {X 0,Y 425.4,Z 140.496,A -85,B 0,C 180,E1 -9707.598,E2 -9707.598} C_VEL
LIN {X 0,Y 425.395,Z 140.497,A -85,B 0,C 180,E1 -9711.449,E2 -9711.449} C_VEL
LIN {X 0,Y 425.497,Z 140.482,A -85,B 0,C 180,E1 -9714.312,E2 -9714.312} C_VEL
LIN {X 0,Y 425.551,Z 140.475,A -85,B 0,C 180,E1 -9718.107,E2 -9718.107} C_VEL
LIN {X 0,Y 425.559,Z 140.474,A -85,B 0,C 180,E1 -9720,E2 -9720} C_VEL
LIN {X 0,Y 425.501,Z 140.483,A -85,B 0,C 180,E1 -9722.84,E2 -9722.84} C_VEL
LIN {X 0,Y 425.516,Z 140.48,A -85,B 0,C 180,E1 -9725.687,E2 -9725.687} C_VEL
LIN {X 0,Y 425.395,Z 140.497,A -85,B 0,C 180,E1 -9728.551,E2 -9728.551} C_VEL
LIN {X 0,Y 425.4,Z 140.496,A -85,B 0,C 180,E1 -9732.402,E2 -9732.402} C_VEL
LIN {X 0,Y 425.375,Z 140.499,A -85,B 0,C 180,E1 -9736.312,E2 -9736.312} C_VEL
LIN {X 0,Y 425.317,Z 140.504,A -85,B 0,C 180,E1 -9739.636,E2 -9739.636} C_VEL
LIN {X 0,Y 425.276,Z 140.511,A -85,B 0,C 180,E1 -9742.339,E2 -9742.339} C_VEL
LIN {X 0,Y 425.308,Z 140.508,A -85,B 0,C 180,E1 -9744.657,E2 -9744.657} C_VEL
LIN {X 0,Y 425.335,Z 140.502,A -85,B 0,C 180,E1 -9747.559,E2 -9747.559} C_VEL
LIN {X 0,Y 425.278,Z 140.512,A -85,B 0,C 180,E1 -9750.817,E2 -9750.817} C_VEL
LIN {X 0,Y 425.3,Z 140.508,A -85,B 0,C 180,E1 -9754.288,E2 -9754.288} C_VEL
LIN {X 0,Y 425.269,Z 140.51,A -85,B 0,C 180,E1 -9757.695,E2 -9757.695} C_VEL
LIN {X 0,Y 425.272,Z 140.513,A -85,B 0,C 180,E1 -9760.521,E2 -9760.521} C_VEL
LIN {X 0,Y 425.249,Z 140.512,A -85,B 0,C 180,E1 -9763.352,E2 -9763.352} C_VEL
LIN {X 0,Y 425.251,Z 140.513,A -85,B 0,C 180,E1 -9766.65,E2 -9766.65} C_VEL
LIN {X 0,Y 425.289,Z 140.509,A -85,B 0,C 180,E1 -9769.875,E2 -9769.875} C_VEL
LIN {X 0,Y 425.273,Z 140.511,A -85,B 0,C 180,E1 -9772.49,E2 -9772.49} C_VEL
LIN {X 0,Y 425.303,Z 140.508,A -85,B 0,C 180,E1 -9775.819,E2 -9775.819} C_VEL
LIN {X 0,Y 425.287,Z 140.506,A -85,B 0,C 180,E1 -9779.24,E2 -9779.24} C_VEL
LIN {X 0,Y 425.411,Z 140.543,A -85,B 0,C 180,E1 -9782.495,E2 -9782.495} C_VEL
LIN {X 0,Y 427.977,Z 154.225,A -85,B 0,C 180,E1 -9785.246,E2 -9785.246} C_VEL
LIN {X 0,Y 427.468,Z 165.643,A -85,B 0,C 180,E1 -9787.368,E2 -9787.368} C_VEL
LIN {X 0,Y 426.412,Z 185.478,A -85,B 0,C 180,E1 -9791.004,E2 -9791.004} C_VEL
LIN {X 0,Y 426.277,Z 188.182,A -85,B 0,C 180,E1 -9791.497,E2 -9791.497} C_VEL
LIN {X 0,Y 429.925,Z 215.193,A -85,B 0,C 180,E1 -9792.11,E2 -9792.11} C_VEL
LIN {X 0,Y 429.146,Z 297.23,A -85,B 0,C 180,E1 -9793.5,E2 -9793.5} C_VEL
LIN {X 0,Y 428.612,Z 310.431,A -85,B 0,C 180,E1 -9793.907,E2 -9793.907} C_VEL
LIN {X 0,Y 428.102,Z 322.588,A -85,B 0,C 180,E1 -9794.468,E2 -9794.468} C_VEL
LIN {X 0,Y 427.369,Z 334.843,A -85,B 0,C 180,E1 -9795.234,E2 -9795.234} C_VEL
LIN {X 0,Y 426.678,Z 346.471,A -85,B 0,C 180,E1 -9796.184,E2 -9796.184} C_VEL
LIN {X 0,Y 426.07,Z 356.937,A -85,B 0,C 180,E1 -9797.256,E2 -9797.256} C_VEL
LIN {X 0,Y 425.553,Z 365.493,A -85,B 0,C 180,E1 -9798.329,E2 -9798.329} C_VEL
LIN {X 0,Y 424.921,Z 374.751,A -85,B 0,C 180,E1 -9799.759,E2 -9799.759} C_VEL
LIN {X 0,Y 424.572,Z 382.204,A -85,B 0,C 180,E1 -9801.193,E2 -9801.193} C_VEL
LIN {X 0,Y 424.331,Z 389.056,A -85,B 0,C 180,E1 -9802.865,E2 -9802.865} C_VEL
LIN {X 0,Y 424.176,Z 393.568,A -85,B 0,C 180,E1 -9804.296,E2 -9804.296} C_VEL
LIN {X 0,Y 424.205,Z 395.951,A -85,B 0,C 180,E1 -9805.249,E2 -9805.249} C_VEL
LIN {X 0,Y 424.13,Z 397.894,A -85,B 0,C 180,E1 -9806.2,E2 -9806.2} C_VEL
LIN {X 0,Y 424.217,Z 399.418,A -85,B 0,C 180,E1 -9807.152,E2 -9807.152} C_VEL
LIN {X 0,Y 424.167,Z 400.479,A -85,B 0,C 180,E1 -9808.102,E2 -9808.102} C_VEL
LIN {X 0,Y 424.142,Z 401.427,A -85,B 0,C 180,E1 -9810.001,E2 -9810.001} C_VEL
LIN {X 0,Y 424.14,Z 401.314,A -85,B 0,C 180,E1 -9810.95,E2 -9810.95} C_VEL
LIN {X 0,Y 424.166,Z 400.767,A -85,B 0,C 180,E1 -9811.9,E2 -9811.9} C_VEL
LIN {X 0,Y 424.178,Z 399.825,A -85,B 0,C 180,E1 -9812.85,E2 -9812.85} C_VEL
LIN {X 0,Y 424.107,Z 398.484,A -85,B 0,C 180,E1 -9813.801,E2 -9813.801} C_VEL
LIN {X 0,Y 424.193,Z 395.66,A -85,B 0,C 180,E1 -9815.229,E2 -9815.229} C_VEL
LIN {X 0,Y 424.225,Z 391.81,A -85,B 0,C 180,E1 -9816.66,E2 -9816.66} C_VEL
LIN {X 0,Y 424.487,Z 386.846,A -85,B 0,C 180,E1 -9818.091,E2 -9818.091} C_VEL
LIN {X 0,Y 424.788,Z 380.612,A -85,B 0,C 180,E1 -9819.524,E2 -9819.524} C_VEL
LIN {X 0,Y 425.32,Z 372.858,A -85,B 0,C 180,E1 -9820.955,E2 -9820.955} C_VEL
LIN {X 0,Y 425.969,Z 364.946,A -85,B 0,C 180,E1 -9822.144,E2 -9822.144} C_VEL
LIN {X 0,Y 426.578,Z 355.306,A -85,B 0,C 180,E1 -9823.336,E2 -9823.336} C_VEL
LIN {X 0,Y 427.359,Z 344.627,A -85,B 0,C 180,E1 -9824.403,E2 -9824.403} C_VEL
LIN {X 0,Y 428.101,Z 334.312,A -85,B 0,C 180,E1 -9825.229,E2 -9825.229} C_VEL
LIN {X 0,Y 428.877,Z 322,A -85,B 0,C 180,E1 -9825.993,E2 -9825.993} C_VEL
LIN {X 0,Y 429.547,Z 309.061,A -85,B 0,C 180,E1 -9826.578,E2 -9826.578} C_VEL
LIN {X 0,Y 430.102,Z 296.511,A -85,B 0,C 180,E1 -9826.953,E2 -9826.953} C_VEL
LIN {X 0,Y 430.974,Z 214.365,A -85,B 0,C 180,E1 -9828.355,E2 -9828.355} C_VEL
LIN {X 0,Y 427.136,Z 190.428,A -85,B 0,C 180,E1 -9828.96,E2 -9828.96} C_VEL
LIN {X 0,Y 426.729,Z 187.895,A -85,B 0,C 180,E1 -9829.047,E2 -9829.047} C_VEL
LIN {X 0,Y 427.886,Z 168.388,A -85,B 0,C 180,E1 -9832.68,E2 -9832.68} C_VEL
LIN {X 0,Y 428.63,Z 157.586,A -85,B 0,C 180,E1 -9834.716,E2 -9834.716} C_VEL
LIN {X 0,Y 427.541,Z 150.811,A -85,B 0,C 180,E1 -9836.1,E2 -9836.1} C_VEL
LIN {X 0,Y 425.338,Z 140.508,A -85,B 0,C 180,E1 -9838.296,E2 -9838.296} C_VEL
LIN {X 0,Y 425.268,Z 140.518,A -85,B 0,C 180,E1 -9841.927,E2 -9841.927} C_VEL
LIN {X 0,Y 425.301,Z 140.507,A -85,B 0,C 180,E1 -9845.336,E2 -9845.336} C_VEL
LIN {X 0,Y 425.294,Z 140.505,A -85,B 0,C 180,E1 -9848.9,E2 -9848.9} C_VEL
LIN {X 0,Y 425.284,Z 140.508,A -85,B 0,C 180,E1 -9851.957,E2 -9851.957} C_VEL
LIN {X 0,Y 425.287,Z 140.512,A -85,B 0,C 180,E1 -9855.283,E2 -9855.283} C_VEL
LIN {X 0,Y 425.258,Z 140.511,A -85,B 0,C 180,E1 -9858.619,E2 -9858.619} C_VEL
LIN {X 0,Y 425.282,Z 140.512,A -85,B 0,C 180,E1 -9861.099,E2 -9861.099} C_VEL
LIN {X 0,Y 425.296,Z 140.508,A -85,B 0,C 180,E1 -9864.664,E2 -9864.664} C_VEL
LIN {X 0,Y 425.264,Z 140.51,A -85,B 0,C 180,E1 -9868.073,E2 -9868.073} C_VEL
LIN {X 0,Y 425.305,Z 140.505,A -85,B 0,C 180,E1 -9871.366,E2 -9871.366} C_VEL
LIN {X 0,Y 425.26,Z 140.513,A -85,B 0,C 180,E1 -9874.552,E2 -9874.552} C_VEL
LIN {X 0,Y 425.291,Z 140.506,A -85,B 0,C 180,E1 -9877.73,E2 -9877.73} C_VEL
LIN {X 0,Y 425.36,Z 140.496,A -85,B 0,C 180,E1 -9880.704,E2 -9880.704} C_VEL
LIN {X 0,Y 425.322,Z 140.502,A -85,B 0,C 180,E1 -9883.686,E2 -9883.686} C_VEL
LIN {X 0,Y 425.407,Z 140.49,A -85,B 0,C 180,E1 -9887.598,E2 -9887.598} C_VEL
LIN {X 0,Y 425.393,Z 140.487,A -85,B 0,C 180,E1 -9891.449,E2 -9891.449} C_VEL
LIN {X 0,Y 425.507,Z 140.483,A -85,B 0,C 180,E1 -9894.313,E2 -9894.313} C_VEL
LIN {X 0,Y 425.563,Z 140.472,A -85,B 0,C 180,E1 -9898.107,E2 -9898.107} C_VEL
LIN {X 0,Y 425.571,Z 140.476,A -85,B 0,C 180,E1 -9900,E2 -9900} C_VEL
LIN {X 0,Y 425.512,Z 140.471,A -85,B 0,C 180,E1 -9902.84,E2 -9902.84} C_VEL
LIN {X 0,Y 425.475,Z 140.482,A -85,B 0,C 180,E1 -9906.48,E2 -9906.48} C_VEL
LIN {X 0,Y 425.396,Z 140.491,A -85,B 0,C 180,E1 -9909.51,E2 -9909.51} C_VEL
LIN {X 0,Y 425.394,Z 140.493,A -85,B 0,C 180,E1 -9912.903,E2 -9912.903} C_VEL
LIN {X 0,Y 425.362,Z 140.497,A -85,B 0,C 180,E1 -9916.604,E2 -9916.604} C_VEL
LIN {X 0,Y 425.329,Z 140.5,A -85,B 0,C 180,E1 -9919.635,E2 -9919.635} C_VEL
LIN {X 0,Y 425.289,Z 140.506,A -85,B 0,C 180,E1 -9922.339,E2 -9922.339} C_VEL
LIN {X 0,Y 425.32,Z 140.5,A -85,B 0,C 180,E1 -9924.657,E2 -9924.657} C_VEL
LIN {X 0,Y 425.301,Z 140.504,A -85,B 0,C 180,E1 -9927.561,E2 -9927.561} C_VEL
LIN {X 0,Y 425.289,Z 140.512,A -85,B 0,C 180,E1 -9930.816,E2 -9930.816} C_VEL
LIN {X 0,Y 425.312,Z 140.505,A -85,B 0,C 180,E1 -9934.288,E2 -9934.288} C_VEL
LIN {X 0,Y 425.28,Z 140.507,A -85,B 0,C 180,E1 -9937.695,E2 -9937.695} C_VEL
LIN {X 0,Y 425.282,Z 140.499,A -85,B 0,C 180,E1 -9940.52,E2 -9940.52} C_VEL
LIN {X 0,Y 425.26,Z 140.51,A -85,B 0,C 180,E1 -9943.351,E2 -9943.351} C_VEL
LIN {X 0,Y 425.259,Z 140.513,A -85,B 0,C 180,E1 -9946.649,E2 -9946.649} C_VEL
LIN {X 0,Y 425.287,Z 140.51,A -85,B 0,C 180,E1 -9949.872,E2 -9949.872} C_VEL
LIN {X 0,Y 425.281,Z 140.51,A -85,B 0,C 180,E1 -9952.489,E2 -9952.489} C_VEL
LIN {X 0,Y 425.311,Z 140.508,A -85,B 0,C 180,E1 -9955.817,E2 -9955.817} C_VEL
LIN {X 0,Y 425.295,Z 140.508,A -85,B 0,C 180,E1 -9959.239,E2 -9959.239} C_VEL
LIN {X 0,Y 425.353,Z 140.504,A -85,B 0,C 180,E1 -9962.442,E2 -9962.442} C_VEL
LIN {X 0,Y 425.407,Z 140.69,A -85,B 0,C 180,E1 -9963.317,E2 -9963.317} C_VEL
LIN {X 0,Y 427.039,Z 149.054,A -85,B 0,C 180,E1 -9965.323,E2 -9965.323} C_VEL
LIN {X 0,Y 427.259,Z 152.152,A -85,B 0,C 180,E1 -9966.029,E2 -9966.029} C_VEL
LIN {X 0,Y 431.428,Z 170.193,A -85,B 0,C 180,E1 -9966.578,E2 -9966.578} C_VEL
LIN {X 0,Y 430.429,Z 259.328,A -85,B 0,C 180,E1 -9968.099,E2 -9968.099} C_VEL
LIN {X 0,Y 429.983,Z 272.943,A -85,B 0,C 180,E1 -9968.526,E2 -9968.526} C_VEL
LIN {X 0,Y 429.51,Z 284.499,A -85,B 0,C 180,E1 -9969.065,E2 -9969.065} C_VEL
LIN {X 0,Y 428.885,Z 297.223,A -85,B 0,C 180,E1 -9969.871,E2 -9969.871} C_VEL
LIN {X 0,Y 428.079,Z 308.813,A -85,B 0,C 180,E1 -9970.831,E2 -9970.831} C_VEL
LIN {X 0,Y 427.411,Z 319.223,A -85,B 0,C 180,E1 -9971.918,E2 -9971.918} C_VEL
LIN {X 0,Y 426.811,Z 327.726,A -85,B 0,C 180,E1 -9973.009,E2 -9973.009} C_VEL
LIN {X 0,Y 426.069,Z 336.834,A -85,B 0,C 180,E1 -9974.451,E2 -9974.451} C_VEL
LIN {X 0,Y 425.442,Z 344.168,A -85,B 0,C 180,E1 -9975.897,E2 -9975.897} C_VEL
LIN {X 0,Y 425.018,Z 349.943,A -85,B 0,C 180,E1 -9977.322,E2 -9977.322} C_VEL
LIN {X 0,Y 424.853,Z 352.177,A -85,B 0,C 180,E1 -9977.978,E2 -9977.978} C_VEL
LIN {X 0,Y 424.026,Z 354.477,A -85,B 0,C 180,E1 -9978.704,E2 -9978.704} C_VEL
LIN {X 0,Y 420.942,Z 357.675,A -85,B 0,C 180,E1 -9979.905,E2 -9979.905} C_VEL
LIN {X 0,Y 417.923,Z 360.227,A -85,B 0,C 180,E1 -9981.155,E2 -9981.155} C_VEL
LIN {X 0,Y 417.213,Z 361.303,A -85,B 0,C 180,E1 -9981.946,E2 -9981.946} C_VEL
LIN {X 0,Y 417.211,Z 362.78,A -85,B 0,C 180,E1 -9983.654,E2 -9983.654} C_VEL
LIN {X 0,Y 417.128,Z 363.032,A -85,B 0,C 180,E1 -9985.167,E2 -9985.167} C_VEL
LIN {X 0,Y 417.192,Z 361.968,A -85,B 0,C 180,E1 -9987.102,E2 -9987.102} C_VEL
LIN {X 0,Y 417.148,Z 360.823,A -85,B 0,C 180,E1 -9988.068,E2 -9988.068} C_VEL
LIN {X 0,Y 417.264,Z 357.298,A -85,B 0,C 180,E1 -9989.999,E2 -9989.999} C_VEL
LIN {X 0,Y 417.449,Z 353.484,A -85,B 0,C 180,E1 -9991.446,E2 -9991.446} C_VEL
LIN {X 0,Y 417.7,Z 348.561,A -85,B 0,C 180,E1 -9992.892,E2 -9992.892} C_VEL
LIN {X 0,Y 418.189,Z 342.368,A -85,B 0,C 180,E1 -9994.336,E2 -9994.336} C_VEL
LIN {X 0,Y 418.745,Z 334.63,A -85,B 0,C 180,E1 -9995.779,E2 -9995.779} C_VEL
LIN {X 0,Y 419.37,Z 326.735,A -85,B 0,C 180,E1 -9996.978,E2 -9996.978} C_VEL
LIN {X 0,Y 420.05,Z 317.115,A -85,B 0,C 180,E1 -9998.175,E2 -9998.175} C_VEL
LIN {X 0,Y 420.779,Z 306.416,A -85,B 0,C 180,E1 -9999.25,E2 -9999.25} C_VEL
LIN {X 0,Y 421.321,Z 295.624,A -85,B 0,C 180,E1 -10000.113,E2 -10000.113} C_VEL
LIN {X 0,Y 421.813,Z 283.496,A -85,B 0,C 180,E1 -10000.863,E2 -10000.863} C_VEL
LIN {X 0,Y 422.232,Z 270.997,A -85,B 0,C 180,E1 -10001.429,E2 -10001.429} C_VEL
LIN {X 0,Y 422.519,Z 257.871,A -85,B 0,C 180,E1 -10001.817,E2 -10001.817} C_VEL
LIN {X 0,Y 423.513,Z 172.419,A -85,B 0,C 180,E1 -10003.273,E2 -10003.273} C_VEL
LIN {X 0,Y 421.208,Z 159.511,A -85,B 0,C 180,E1 -10003.593,E2 -10003.593} C_VEL
LIN {X 0,Y 419.774,Z 152.352,A -85,B 0,C 180,E1 -10003.785,E2 -10003.785} C_VEL
LIN {X 0,Y 419.603,Z 147.843,A -85,B 0,C 180,E1 -10004.798,E2 -10004.798} C_VEL
LIN {X 0,Y 418.373,Z 141.374,A -85,B 0,C 180,E1 -10006.341,E2 -10006.341} C_VEL
LIN {X 0,Y 418.271,Z 141.384,A -85,B 0,C 180,E1 -10009.789,E2 -10009.789} C_VEL
LIN {X 0,Y 418.232,Z 141.387,A -85,B 0,C 180,E1 -10012.735,E2 -10012.735} C_VEL
LIN {X 0,Y 418.267,Z 141.384,A -85,B 0,C 180,E1 -10015.903,E2 -10015.903} C_VEL
LIN {X 0,Y 418.263,Z 141.381,A -85,B 0,C 180,E1 -10019.161,E2 -10019.161} C_VEL
LIN {X 0,Y 418.255,Z 141.383,A -85,B 0,C 180,E1 -10022.843,E2 -10022.843} C_VEL
LIN {X 0,Y 418.241,Z 141.388,A -85,B 0,C 180,E1 -10026.237,E2 -10026.237} C_VEL
LIN {X 0,Y 418.25,Z 141.387,A -85,B 0,C 180,E1 -10029.68,E2 -10029.68} C_VEL
LIN {X 0,Y 418.225,Z 141.389,A -85,B 0,C 180,E1 -10032.32,E2 -10032.32} C_VEL
LIN {X 0,Y 418.23,Z 141.387,A -85,B 0,C 180,E1 -10035.107,E2 -10035.107} C_VEL
LIN {X 0,Y 418.233,Z 141.39,A -85,B 0,C 180,E1 -10037.766,E2 -10037.766} C_VEL
LIN {X 0,Y 418.238,Z 141.386,A -85,B 0,C 180,E1 -10040.62,E2 -10040.62} C_VEL
LIN {X 0,Y 418.234,Z 141.388,A -85,B 0,C 180,E1 -10043.975,E2 -10043.975} C_VEL
LIN {X 0,Y 418.248,Z 141.386,A -85,B 0,C 180,E1 -10047.155,E2 -10047.155} C_VEL
LIN {X 0,Y 418.259,Z 141.384,A -85,B 0,C 180,E1 -10050.895,E2 -10050.895} C_VEL
LIN {X 0,Y 418.249,Z 141.386,A -85,B 0,C 180,E1 -10054.094,E2 -10054.094} C_VEL
LIN {X 0,Y 418.22,Z 141.392,A -85,B 0,C 180,E1 -10057.263,E2 -10057.263} C_VEL
LIN {X 0,Y 418.272,Z 141.382,A -85,B 0,C 180,E1 -10060.363,E2 -10060.363} C_VEL
LIN {X 0,Y 418.304,Z 141.38,A -85,B 0,C 180,E1 -10063.404,E2 -10063.404} C_VEL
LIN {X 0,Y 418.335,Z 141.377,A -85,B 0,C 180,E1 -10066.999,E2 -10066.999} C_VEL
LIN {X 0,Y 418.325,Z 141.375,A -85,B 0,C 180,E1 -10070.328,E2 -10070.328} C_VEL
LIN {X 0,Y 418.429,Z 141.365,A -85,B 0,C 180,E1 -10073.248,E2 -10073.248} C_VEL
LIN {X 0,Y 418.302,Z 141.38,A -85,B 0,C 180,E1 -10075.181,E2 -10075.181} C_VEL
LIN {X 0,Y 418.52,Z 141.351,A -85,B 0,C 180,E1 -10078.075,E2 -10078.075} C_VEL
LIN {X 0,Y 418.393,Z 141.369,A -85,B 0,C 180,E1 -10080.962,E2 -10080.962} C_VEL
LIN {X 0,Y 418.458,Z 141.361,A -85,B 0,C 180,E1 -10082.888,E2 -10082.888} C_VEL
LIN {X 0,Y 418.473,Z 141.357,A -85,B 0,C 180,E1 -10085.783,E2 -10085.783} C_VEL
LIN {X 0,Y 418.365,Z 141.372,A -85,B 0,C 180,E1 -10088.696,E2 -10088.696} C_VEL
LIN {X 0,Y 418.301,Z 141.378,A -85,B 0,C 180,E1 -10091.631,E2 -10091.631} C_VEL
LIN {X 0,Y 418.287,Z 141.382,A -85,B 0,C 180,E1 -10094.598,E2 -10094.598} C_VEL
LIN {X 0,Y 418.267,Z 141.382,A -85,B 0,C 180,E1 -10097.605,E2 -10097.605} C_VEL
LIN {X 0,Y 418.238,Z 141.389,A -85,B 0,C 180,E1 -10100.664,E2 -10100.664} C_VEL
LIN {X 0,Y 418.261,Z 141.383,A -85,B 0,C 180,E1 -10103.783,E2 -10103.783} C_VEL
LIN {X 0,Y 418.3,Z 141.379,A -85,B 0,C 180,E1 -10107.071,E2 -10107.071} C_VEL
LIN {X 0,Y 418.234,Z 141.388,A -85,B 0,C 180,E1 -10110.273,E2 -10110.273} C_VEL
LIN {X 0,Y 418.238,Z 141.386,A -85,B 0,C 180,E1 -10113.678,E2 -10113.678} C_VEL
LIN {X 0,Y 418.231,Z 141.386,A -85,B 0,C 180,E1 -10117.225,E2 -10117.225} C_VEL
LIN {X 0,Y 418.236,Z 141.386,A -85,B 0,C 180,E1 -10119.684,E2 -10119.684} C_VEL
LIN {X 0,Y 418.222,Z 141.392,A -85,B 0,C 180,E1 -10122.322,E2 -10122.322} C_VEL
LIN {X 0,Y 418.229,Z 141.386,A -85,B 0,C 180,E1 -10125.11,E2 -10125.11} C_VEL
LIN {X 0,Y 418.234,Z 141.387,A -85,B 0,C 180,E1 -10127.768,E2 -10127.768} C_VEL
LIN {X 0,Y 418.253,Z 141.384,A -85,B 0,C 180,E1 -10130.62,E2 -10130.62} C_VEL
LIN {X 0,Y 418.238,Z 141.389,A -85,B 0,C 180,E1 -10133.977,E2 -10133.977} C_VEL
LIN {X 0,Y 418.254,Z 141.382,A -85,B 0,C 180,E1 -10137.157,E2 -10137.157} C_VEL
LIN {X 0,Y 418.265,Z 141.385,A -85,B 0,C 180,E1 -10140.897,E2 -10140.897} C_VEL
LIN {X 0,Y 418.354,Z 141.453,A -85,B 0,C 180,E1 -10142.274,E2 -10142.274} C_VEL
LIN {X 0,Y 420.995,Z 155.282,A -85,B 0,C 180,E1 -10145.108,E2 -10145.108} C_VEL
LIN {X 0,Y 420.648,Z 164.039,A -85,B 0,C 180,E1 -10146.768,E2 -10146.768} C_VEL
LIN {X 0,Y 419.557,Z 183.634,A -85,B 0,C 180,E1 -10150.427,E2 -10150.427} C_VEL
LIN {X 0,Y 419.295,Z 187.855,A -85,B 0,C 180,E1 -10151.209,E2 -10151.209} C_VEL
